LIN {X 0,Y 549.651,Z 687.436,A -85,B 0,C 180,E1 21205.612,E2 21205.612} C_VEL
LIN {X 0,Y 543.222,Z 825.686,A -85,B 0,C 180,E1 21203.522,E2 21203.522} C_VEL
LIN {X 0,Y 540.973,Z 851.994,A -85,B 0,C 180,E1 21203.026,E2 21203.026} C_VEL
LIN {X 0,Y 537.634,Z 879.368,A -85,B 0,C 180,E1 21202.319,E2 21202.319} C_VEL
LIN {X 0,Y 534.444,Z 901.056,A -85,B 0,C 180,E1 21201.617,E2 21201.617} C_VEL
LIN {X 0,Y 531.01,Z 921.384,A -85,B 0,C 180,E1 21200.832,E2 21200.832} C_VEL
LIN {X 0,Y 527.002,Z 942.572,A -85,B 0,C 180,E1 21199.871,E2 21199.871} C_VEL
LIN {X 0,Y 521.583,Z 968.283,A -85,B 0,C 180,E1 21198.494,E2 21198.494} C_VEL
LIN {X 0,Y 516.27,Z 990.784,A -85,B 0,C 180,E1 21197.06,E2 21197.06} C_VEL
LIN {X 0,Y 511.706,Z 1008.978,A -85,B 0,C 180,E1 21195.736,E2 21195.736} C_VEL
LIN {X 0,Y 507.179,Z 1026.1,A -85,B 0,C 180,E1 21194.336,E2 21194.336} C_VEL
LIN {X 0,Y 502.54,Z 1042.949,A -85,B 0,C 180,E1 21192.793,E2 21192.793} C_VEL
LIN {X 0,Y 497.445,Z 1060.954,A -85,B 0,C 180,E1 21190.939,E2 21190.939} C_VEL
LIN {X 0,Y 491.162,Z 1082.539,A -85,B 0,C 180,E1 21188.381,E2 21188.381} C_VEL
LIN {X 0,Y 486.635,Z 1097.975,A -85,B 0,C 180,E1 21186.28,E2 21186.28} C_VEL
LIN {X 0,Y 482.591,Z 1111.902,A -85,B 0,C 180,E1 21184.158,E2 21184.158} C_VEL
LIN {X 0,Y 479.016,Z 1124.472,A -85,B 0,C 180,E1 21182.017,E2 21182.017} C_VEL
LIN {X 0,Y 475.599,Z 1137.117,A -85,B 0,C 180,E1 21179.607,E2 21179.607} C_VEL
LIN {X 0,Y 472.036,Z 1151.255,A -85,B 0,C 180,E1 21176.547,E2 21176.547} C_VEL
LIN {X 0,Y 469.365,Z 1162.835,A -85,B 0,C 180,E1 21173.608,E2 21173.608} C_VEL
LIN {X 0,Y 467.505,Z 1172.064,A -85,B 0,C 180,E1 21170.926,E2 21170.926} C_VEL
LIN {X 0,Y 466.177,Z 1179.694,A -85,B 0,C 180,E1 21168.378,E2 21168.378} C_VEL
LIN {X 0,Y 465.207,Z 1186.55,A -85,B 0,C 180,E1 21165.712,E2 21165.712} C_VEL
LIN {X 0,Y 464.466,Z 1193.301,A -85,B 0,C 180,E1 21162.558,E2 21162.558} C_VEL
LIN {X 0,Y 464.091,Z 1198.542,A -85,B 0,C 180,E1 21159.299,E2 21159.299} C_VEL
LIN {X 0,Y 463.959,Z 1201.757,A -85,B 0,C 180,E1 21156.527,E2 21156.527} C_VEL
LIN {X 0,Y 463.915,Z 1203.743,A -85,B 0,C 180,E1 21153.955,E2 21153.955} C_VEL
LIN {X 0,Y 463.911,Z 1204.734,A -85,B 0,C 180,E1 21151.482,E2 21151.482} C_VEL
LIN {X 0,Y 463.908,Z 1204.825,A -85,B 0,C 180,E1 21149.012,E2 21149.012} C_VEL
LIN {X 0,Y 463.915,Z 1204.015,A -85,B 0,C 180,E1 21146.54,E2 21146.54} C_VEL
LIN {X 0,Y 463.947,Z 1202.181,A -85,B 0,C 180,E1 21143.938,E2 21143.938} C_VEL
LIN {X 0,Y 464.044,Z 1199.499,A -85,B 0,C 180,E1 21141.45,E2 21141.45} C_VEL
LIN {X 0,Y 464.248,Z 1195.868,A -85,B 0,C 180,E1 21138.949,E2 21138.949} C_VEL
LIN {X 0,Y 464.693,Z 1190.99,A -85,B 0,C 180,E1 21136.309,E2 21136.309} C_VEL
LIN {X 0,Y 465.387,Z 1185.014,A -85,B 0,C 180,E1 21133.653,E2 21133.653} C_VEL
LIN {X 0,Y 466.671,Z 1176.831,A -85,B 0,C 180,E1 21130.604,E2 21130.604} C_VEL
LIN {X 0,Y 468.694,Z 1166.058,A -85,B 0,C 180,E1 21127.287,E2 21127.287} C_VEL
LIN {X 0,Y 470.899,Z 1155.903,A -85,B 0,C 180,E1 21124.602,E2 21124.602} C_VEL
LIN {X 0,Y 473.407,Z 1145.514,A -85,B 0,C 180,E1 21122.176,E2 21122.176} C_VEL
LIN {X 0,Y 476.604,Z 1133.238,A -85,B 0,C 180,E1 21119.63,E2 21119.63} C_VEL
LIN {X 0,Y 481.3,Z 1116.533,A -85,B 0,C 180,E1 21116.598,E2 21116.598} C_VEL
LIN {X 0,Y 485.893,Z 1100.648,A -85,B 0,C 180,E1 21114.094,E2 21114.094} C_VEL
LIN {X 0,Y 490.368,Z 1085.693,A -85,B 0,C 180,E1 21111.992,E2 21111.992} C_VEL
LIN {X 0,Y 495.392,Z 1069.058,A -85,B 0,C 180,E1 21109.904,E2 21109.904} C_VEL
LIN {X 0,Y 501.937,Z 1047.349,A -85,B 0,C 180,E1 21107.524,E2 21107.524} C_VEL
LIN {X 0,Y 507.495,Z 1028.134,A -85,B 0,C 180,E1 21105.699,E2 21105.699} C_VEL
LIN {X 0,Y 512.508,Z 1010.266,A -85,B 0,C 180,E1 21104.196,E2 21104.196} C_VEL
LIN {X 0,Y 517.402,Z 991.974,A -85,B 0,C 180,E1 21102.831,E2 21102.831} C_VEL
LIN {X 0,Y 522.564,Z 971.525,A -85,B 0,C 180,E1 21101.489,E2 21101.489} C_VEL
LIN {X 0,Y 528.704,Z 945.004,A -85,B 0,C 180,E1 21100.012,E2 21100.012} C_VEL
LIN {X 0,Y 533.198,Z 923.023,A -85,B 0,C 180,E1 21098.988,E2 21098.988} C_VEL
LIN {X 0,Y 536.991,Z 902.347,A -85,B 0,C 180,E1 21098.171,E2 21098.171} C_VEL
LIN {X 0,Y 540.352,Z 881.367,A -85,B 0,C 180,E1 21097.475,E2 21097.475} C_VEL
LIN {X 0,Y 543.373,Z 859.139,A -85,B 0,C 180,E1 21096.872,E2 21096.872} C_VEL
LIN {X 0,Y 546.347,Z 831.001,A -85,B 0,C 180,E1 21096.29,E2 21096.29} C_VEL
LIN {X 0,Y 549.102,Z 782.806,A -85,B 0,C 180,E1 21095.529,E2 21095.529} C_VEL
LIN {X 0,Y 560.963,Z 560.073,A -85,B 0,C 180,E1 21092.109,E2 21092.109} C_VEL
LIN {X 0,Y 565.673,Z 475.855,A -85,B 0,C 180,E1 21090.8,E2 21090.8} C_VEL
LIN {X 0,Y 556.142,Z 460.846,A -85,B 0,C 180,E1 21088.483,E2 21088.483} C_VEL
LIN {X 0,Y 548.365,Z 449.512,A -85,B 0,C 180,E1 21086.389,E2 21086.389} C_VEL
LIN {X 0,Y 541.388,Z 439.723,A -85,B 0,C 180,E1 21084.293,E2 21084.293} C_VEL
LIN {X 0,Y 536.871,Z 433.476,A -85,B 0,C 180,E1 21082.792,E2 21082.792} C_VEL
LIN {X 0,Y 532.572,Z 428.076,A -85,B 0,C 180,E1 21081.245,E2 21081.245} C_VEL
LIN {X 0,Y 528.819,Z 423.299,A -85,B 0,C 180,E1 21079.754,E2 21079.754} C_VEL
LIN {X 0,Y 524.766,Z 418.77,A -85,B 0,C 180,E1 21077.979,E2 21077.979} C_VEL
LIN {X 0,Y 523.478,Z 416.816,A -85,B 0,C 180,E1 21077.336,E2 21077.336} C_VEL
LIN {X 0,Y 519.967,Z 413.289,A -85,B 0,C 180,E1 21075.503,E2 21075.503} C_VEL
LIN {X 0,Y 518.406,Z 410.788,A -85,B 0,C 180,E1 21074.521,E2 21074.521} C_VEL
LIN {X 0,Y 515.036,Z 407.8,A -85,B 0,C 180,E1 21072.217,E2 21072.217} C_VEL
LIN {X 0,Y 513.302,Z 404.463,A -85,B 0,C 180,E1 21070.551,E2 21070.551} C_VEL
LIN {X 0,Y 509.592,Z 401.905,A -85,B 0,C 180,E1 21064.276,E2 21064.276} C_VEL
LIN {X 0,Y 509.876,Z 402.177,A -85,B 0,C 180,E1 21061.236,E2 21061.236} C_VEL
LIN {X 0,Y 513.509,Z 404.739,A -85,B 0,C 180,E1 21056.036,E2 21056.036} C_VEL
LIN {X 0,Y 515.352,Z 408.233,A -85,B 0,C 180,E1 21054.321,E2 21054.321} C_VEL
LIN {X 0,Y 518.812,Z 411.217,A -85,B 0,C 180,E1 21052.024,E2 21052.024} C_VEL
LIN {X 0,Y 521.465,Z 415.141,A -85,B 0,C 180,E1 21050.453,E2 21050.453} C_VEL
LIN {X 0,Y 524.069,Z 417.551,A -85,B 0,C 180,E1 21049.168,E2 21049.168} C_VEL
LIN {X 0,Y 527.266,Z 421.812,A -85,B 0,C 180,E1 21047.682,E2 21047.682} C_VEL
LIN {X 0,Y 529.035,Z 423.657,A -85,B 0,C 180,E1 21046.947,E2 21046.947} C_VEL
LIN {X 0,Y 532.738,Z 428.24,A -85,B 0,C 180,E1 21045.489,E2 21045.489} C_VEL
LIN {X 0,Y 538.696,Z 435.728,A -85,B 0,C 180,E1 21043.391,E2 21043.391} C_VEL
LIN {X 0,Y 543.283,Z 441.609,A -85,B 0,C 180,E1 21041.934,E2 21041.934} C_VEL
LIN {X 0,Y 549.857,Z 450.066,A -85,B 0,C 180,E1 21040.037,E2 21040.037} C_VEL
LIN {X 0,Y 559.197,Z 463.027,A -85,B 0,C 180,E1 21037.613,E2 21037.613} C_VEL
LIN {X 0,Y 565.694,Z 473.379,A -85,B 0,C 180,E1 21036.056,E2 21036.056} C_VEL
LIN {X 0,Y 553.81,Z 688.927,A -85,B 0,C 180,E1 21032.734,E2 21032.734} C_VEL
LIN {X 0,Y 546.853,Z 819.072,A -85,B 0,C 180,E1 21030.725,E2 21030.725} C_VEL
LIN {X 0,Y 544.343,Z 846.185,A -85,B 0,C 180,E1 21030.201,E2 21030.201} C_VEL
LIN {X 0,Y 540.821,Z 872.767,A -85,B 0,C 180,E1 21029.495,E2 21029.495} C_VEL
LIN {X 0,Y 537.599,Z 893.258,A -85,B 0,C 180,E1 21028.819,E2 21028.819} C_VEL
LIN {X 0,Y 533.943,Z 913.499,A -85,B 0,C 180,E1 21028.025,E2 21028.025} C_VEL
LIN {X 0,Y 529.736,Z 934.282,A -85,B 0,C 180,E1 21027.07,E2 21027.07} C_VEL
LIN {X 0,Y 524.349,Z 958.432,A -85,B 0,C 180,E1 21025.768,E2 21025.768} C_VEL
LIN {X 0,Y 518.322,Z 982.281,A -85,B 0,C 180,E1 21024.231,E2 21024.231} C_VEL
LIN {X 0,Y 513.236,Z 1001.222,A -85,B 0,C 180,E1 21022.824,E2 21022.824} C_VEL
LIN {X 0,Y 508.27,Z 1018.81,A -85,B 0,C 180,E1 21021.349,E2 21021.349} C_VEL
LIN {X 0,Y 503.044,Z 1036.665,A -85,B 0,C 180,E1 21019.663,E2 21019.663} C_VEL
LIN {X 0,Y 496.66,Z 1057.893,A -85,B 0,C 180,E1 21017.376,E2 21017.376} C_VEL
LIN {X 0,Y 491.067,Z 1075.973,A -85,B 0,C 180,E1 21015.118,E2 21015.118} C_VEL
LIN {X 0,Y 486.515,Z 1090.867,A -85,B 0,C 180,E1 21013.024,E2 21013.024} C_VEL
LIN {X 0,Y 482.248,Z 1105.162,A -85,B 0,C 180,E1 21010.775,E2 21010.775} C_VEL
LIN {X 0,Y 477.553,Z 1121.65,A -85,B 0,C 180,E1 21007.84,E2 21007.84} C_VEL
LIN {X 0,Y 475.09,Z 1130.636,A -85,B 0,C 180,E1 21006.035,E2 21006.035} C_VEL
LIN {X 0,Y 473.128,Z 1134.565,A -85,B 0,C 180,E1 21005.261,E2 21005.261} C_VEL
LIN {X 0,Y 464.651,Z 1144.816,A -85,B 0,C 180,E1 21003.232,E2 21003.232} C_VEL
LIN {X 0,Y 463.204,Z 1147.79,A -85,B 0,C 180,E1 21002.52,E2 21002.52} C_VEL
LIN {X 0,Y 460.393,Z 1159.963,A -85,B 0,C 180,E1 20999.109,E2 20999.109} C_VEL
LIN {X 0,Y 458.412,Z 1169.958,A -85,B 0,C 180,E1 20995.725,E2 20995.725} C_VEL
LIN {X 0,Y 457.267,Z 1177.255,A -85,B 0,C 180,E1 20992.77,E2 20992.77} C_VEL
LIN {X 0,Y 456.495,Z 1183.735,A -85,B 0,C 180,E1 20989.579,E2 20989.579} C_VEL
LIN {X 0,Y 456.092,Z 1188.961,A -85,B 0,C 180,E1 20986.165,E2 20986.165} C_VEL
LIN {X 0,Y 455.953,Z 1192.065,A -85,B 0,C 180,E1 20983.312,E2 20983.312} C_VEL
LIN {X 0,Y 455.916,Z 1193.909,A -85,B 0,C 180,E1 20980.724,E2 20980.724} C_VEL
LIN {X 0,Y 455.908,Z 1194.803,A -85,B 0,C 180,E1 20978.196,E2 20978.196} C_VEL
LIN {X 0,Y 455.911,Z 1194.794,A -85,B 0,C 180,E1 20975.664,E2 20975.664} C_VEL
LIN {X 0,Y 455.916,Z 1193.822,A -85,B 0,C 180,E1 20973.017,E2 20973.017} C_VEL
LIN {X 0,Y 455.974,Z 1191.657,A -85,B 0,C 180,E1 20970.126,E2 20970.126} C_VEL
LIN {X 0,Y 456.177,Z 1187.597,A -85,B 0,C 180,E1 20966.733,E2 20966.733} C_VEL
LIN {X 0,Y 456.608,Z 1182.552,A -85,B 0,C 180,E1 20963.714,E2 20963.714} C_VEL
LIN {X 0,Y 457.356,Z 1176.516,A -85,B 0,C 180,E1 20960.817,E2 20960.817} C_VEL
LIN {X 0,Y 458.685,Z 1168.537,A -85,B 0,C 180,E1 20957.665,E2 20957.665} C_VEL
LIN {X 0,Y 460.867,Z 1157.701,A -85,B 0,C 180,E1 20954.136,E2 20954.136} C_VEL
LIN {X 0,Y 463.467,Z 1146.69,A -85,B 0,C 180,E1 20951.119,E2 20951.119} C_VEL
LIN {X 0,Y 466.481,Z 1135.156,A -85,B 0,C 180,E1 20948.367,E2 20948.367} C_VEL
LIN {X 0,Y 470.784,Z 1120.249,A -85,B 0,C 180,E1 20945.267,E2 20945.267} C_VEL
LIN {X 0,Y 475.265,Z 1105.063,A -85,B 0,C 180,E1 20942.566,E2 20942.566} C_VEL
LIN {X 0,Y 479.518,Z 1091.202,A -85,B 0,C 180,E1 20940.385,E2 20940.385} C_VEL
LIN {X 0,Y 484.266,Z 1075.83,A -85,B 0,C 180,E1 20938.231,E2 20938.231} C_VEL
LIN {X 0,Y 490.176,Z 1056.8,A -85,B 0,C 180,E1 20935.879,E2 20935.879} C_VEL
LIN {X 0,Y 496.306,Z 1036.036,A -85,B 0,C 180,E1 20933.68,E2 20933.68} C_VEL
LIN {X 0,Y 501.213,Z 1018.99,A -85,B 0,C 180,E1 20932.09,E2 20932.09} C_VEL
LIN {X 0,Y 506.037,Z 1001.468,A -85,B 0,C 180,E1 20930.636,E2 20930.636} C_VEL
LIN {X 0,Y 510.938,Z 982.649,A -85,B 0,C 180,E1 20929.253,E2 20929.253} C_VEL
LIN {X 0,Y 516.7,Z 959.081,A -85,B 0,C 180,E1 20927.744,E2 20927.744} C_VEL
LIN {X 0,Y 521.835,Z 935.199,A -85,B 0,C 180,E1 20926.464,E2 20926.464} C_VEL
LIN {X 0,Y 525.854,Z 914.588,A -85,B 0,C 180,E1 20925.52,E2 20925.52} C_VEL
LIN {X 0,Y 529.423,Z 894.057,A -85,B 0,C 180,E1 20924.718,E2 20924.718} C_VEL
LIN {X 0,Y 532.612,Z 872.81,A -85,B 0,C 180,E1 20924.019,E2 20924.019} C_VEL
LIN {X 0,Y 535.973,Z 846.163,A -85,B 0,C 180,E1 20923.314,E2 20923.314} C_VEL
LIN {X 0,Y 538.366,Z 818.867,A -85,B 0,C 180,E1 20922.792,E2 20922.792} C_VEL
LIN {X 0,Y 544.33,Z 695.866,A -85,B 0,C 180,E1 20920.922,E2 20920.922} C_VEL
LIN {X 0,Y 555.064,Z 476.693,A -85,B 0,C 180,E1 20917.593,E2 20917.593} C_VEL
LIN {X 0,Y 554.881,Z 475.782,A -85,B 0,C 180,E1 20917.543,E2 20917.543} C_VEL
LIN {X 0,Y 544.972,Z 460.83,A -85,B 0,C 180,E1 20915.532,E2 20915.532} C_VEL
LIN {X 0,Y 533.991,Z 445.737,A -85,B 0,C 180,E1 20913.114,E2 20913.114} C_VEL
LIN {X 0,Y 525.45,Z 434.579,A -85,B 0,C 180,E1 20911.044,E2 20911.044} C_VEL
LIN {X 0,Y 518.137,Z 425.158,A -85,B 0,C 180,E1 20909.098,E2 20909.098} C_VEL
LIN {X 0,Y 513.762,Z 419.766,A -85,B 0,C 180,E1 20907.846,E2 20907.846} C_VEL
LIN {X 0,Y 509.435,Z 414.406,A -85,B 0,C 180,E1 20906.521,E2 20906.521} C_VEL
LIN {X 0,Y 504.85,Z 408.87,A -85,B 0,C 180,E1 20905.015,E2 20905.015} C_VEL
LIN {X 0,Y 501.142,Z 404.499,A -85,B 0,C 180,E1 20903.7,E2 20903.7} C_VEL
LIN {X 0,Y 499.827,Z 402.982,A -85,B 0,C 180,E1 20903.21,E2 20903.21} C_VEL
LIN {X 0,Y 496.356,Z 399.083,A -85,B 0,C 180,E1 20901.85,E2 20901.85} C_VEL
LIN {X 0,Y 495.128,Z 397.19,A -85,B 0,C 180,E1 20901.316,E2 20901.316} C_VEL
LIN {X 0,Y 491.632,Z 393.913,A -85,B 0,C 180,E1 20899.794,E2 20899.794} C_VEL
LIN {X 0,Y 489.71,Z 390.934,A -85,B 0,C 180,E1 20898.821,E2 20898.821} C_VEL
LIN {X 0,Y 486.447,Z 388.452,A -85,B 0,C 180,E1 20897.155,E2 20897.155} C_VEL
LIN {X 0,Y 484.363,Z 384.721,A -85,B 0,C 180,E1 20895.813,E2 20895.813} C_VEL
LIN {X 0,Y 480.409,Z 381.967,A -85,B 0,C 180,E1 20893.113,E2 20893.113} C_VEL
LIN {X 0,Y 478.502,Z 378.278,A -85,B 0,C 180,E1 20891.206,E2 20891.206} C_VEL
LIN {X 0,Y 478.048,Z 377.801,A -85,B 0,C 180,E1 20890.728,E2 20890.728} C_VEL
LIN {X 0,Y 474.633,Z 375.968,A -85,B 0,C 180,E1 20884.228,E2 20884.228} C_VEL
LIN {X 0,Y 475.297,Z 376.512,A -85,B 0,C 180,E1 20880.241,E2 20880.241} C_VEL
LIN {X 0,Y 478.483,Z 378.16,A -85,B 0,C 180,E1 20875.926,E2 20875.926} C_VEL
LIN {X 0,Y 480.364,Z 381.936,A -85,B 0,C 180,E1 20874.026,E2 20874.026} C_VEL
LIN {X 0,Y 484.421,Z 384.931,A -85,B 0,C 180,E1 20871.244,E2 20871.244} C_VEL
LIN {X 0,Y 486.469,Z 388.438,A -85,B 0,C 180,E1 20869.938,E2 20869.938} C_VEL
LIN {X 0,Y 490.121,Z 391.389,A -85,B 0,C 180,E1 20868.079,E2 20868.079} C_VEL
LIN {X 0,Y 492.974,Z 395.508,A -85,B 0,C 180,E1 20866.69,E2 20866.69} C_VEL
LIN {X 0,Y 495.56,Z 397.796,A -85,B 0,C 180,E1 20865.6,E2 20865.6} C_VEL
LIN {X 0,Y 498.739,Z 402.022,A -85,B 0,C 180,E1 20864.297,E2 20864.297} C_VEL
LIN {X 0,Y 500.891,Z 404.06,A -85,B 0,C 180,E1 20863.503,E2 20863.503} C_VEL
LIN {X 0,Y 504.6,Z 408.613,A -85,B 0,C 180,E1 20862.173,E2 20862.173} C_VEL
LIN {X 0,Y 506.266,Z 410.618,A -85,B 0,C 180,E1 20861.608,E2 20861.608} C_VEL
LIN {X 0,Y 511.081,Z 416.441,A -85,B 0,C 180,E1 20860.068,E2 20860.068} C_VEL
LIN {X 0,Y 516.19,Z 422.736,A -85,B 0,C 180,E1 20858.554,E2 20858.554} C_VEL
LIN {X 0,Y 521.204,Z 429.022,A -85,B 0,C 180,E1 20857.17,E2 20857.17} C_VEL
LIN {X 0,Y 528.614,Z 439.045,A -85,B 0,C 180,E1 20855.26,E2 20855.26} C_VEL
LIN {X 0,Y 539.958,Z 455.564,A -85,B 0,C 180,E1 20852.602,E2 20852.602} C_VEL
LIN {X 0,Y 552.93,Z 475.552,A -85,B 0,C 180,E1 20849.88,E2 20849.88} C_VEL
LIN {X 0,Y 555.066,Z 479.191,A -85,B 0,C 180,E1 20849.453,E2 20849.453} C_VEL
LIN {X 0,Y 544.676,Z 691.913,A -85,B 0,C 180,E1 20846.221,E2 20846.221} C_VEL
LIN {X 0,Y 538.232,Z 825.714,A -85,B 0,C 180,E1 20844.188,E2 20844.188} C_VEL
LIN {X 0,Y 535.869,Z 852.634,A -85,B 0,C 180,E1 20843.678,E2 20843.678} C_VEL
LIN {X 0,Y 532.469,Z 879.552,A -85,B 0,C 180,E1 20842.978,E2 20842.978} C_VEL
LIN {X 0,Y 529.193,Z 901.157,A -85,B 0,C 180,E1 20842.276,E2 20842.276} C_VEL
LIN {X 0,Y 525.597,Z 921.833,A -85,B 0,C 180,E1 20841.474,E2 20841.474} C_VEL
LIN {X 0,Y 521.474,Z 942.982,A -85,B 0,C 180,E1 20840.51,E2 20840.51} C_VEL
LIN {X 0,Y 515.816,Z 968.907,A -85,B 0,C 180,E1 20839.11,E2 20839.11} C_VEL
LIN {X 0,Y 510.472,Z 990.866,A -85,B 0,C 180,E1 20837.702,E2 20837.702} C_VEL
LIN {X 0,Y 505.707,Z 1009.256,A -85,B 0,C 180,E1 20836.355,E2 20836.355} C_VEL
LIN {X 0,Y 501.026,Z 1026.358,A -85,B 0,C 180,E1 20834.947,E2 20834.947} C_VEL
LIN {X 0,Y 495.943,Z 1044.189,A -85,B 0,C 180,E1 20833.295,E2 20833.295} C_VEL
LIN {X 0,Y 489.829,Z 1065.1,A -85,B 0,C 180,E1 20831.092,E2 20831.092} C_VEL
LIN {X 0,Y 483.991,Z 1084.163,A -85,B 0,C 180,E1 20828.752,E2 20828.752} C_VEL
LIN {X 0,Y 479.602,Z 1098.623,A -85,B 0,C 180,E1 20826.75,E2 20826.75} C_VEL
LIN {X 0,Y 475.404,Z 1112.517,A -85,B 0,C 180,E1 20824.601,E2 20824.601} C_VEL
LIN {X 0,Y 471.263,Z 1126.56,A -85,B 0,C 180,E1 20822.159,E2 20822.159} C_VEL
LIN {X 0,Y 466.786,Z 1142.559,A -85,B 0,C 180,E1 20818.953,E2 20818.953} C_VEL
LIN {X 0,Y 463.732,Z 1154.271,A -85,B 0,C 180,E1 20816.232,E2 20816.232} C_VEL
LIN {X 0,Y 461.405,Z 1164.129,A -85,B 0,C 180,E1 20813.634,E2 20813.634} C_VEL
LIN {X 0,Y 459.589,Z 1172.789,A -85,B 0,C 180,E1 20811.037,E2 20811.037} C_VEL
LIN {X 0,Y 458.102,Z 1181.027,A -85,B 0,C 180,E1 20808.187,E2 20808.187} C_VEL
LIN {X 0,Y 456.901,Z 1189.62,A -85,B 0,C 180,E1 20804.576,E2 20804.576} C_VEL
LIN {X 0,Y 456.323,Z 1195.154,A -85,B 0,C 180,E1 20801.629,E2 20801.629} C_VEL
LIN {X 0,Y 456.077,Z 1198.95,A -85,B 0,C 180,E1 20799.082,E2 20799.082} C_VEL
LIN {X 0,Y 455.96,Z 1201.798,A -85,B 0,C 180,E1 20796.548,E2 20796.548} C_VEL
LIN {X 0,Y 455.915,Z 1203.718,A -85,B 0,C 180,E1 20794.024,E2 20794.024} C_VEL
LIN {X 0,Y 455.91,Z 1204.722,A -85,B 0,C 180,E1 20791.508,E2 20791.508} C_VEL
LIN {X 0,Y 455.908,Z 1204.814,A -85,B 0,C 180,E1 20788.995,E2 20788.995} C_VEL
LIN {X 0,Y 455.915,Z 1203.992,A -85,B 0,C 180,E1 20786.479,E2 20786.479} C_VEL
LIN {X 0,Y 455.946,Z 1202.255,A -85,B 0,C 180,E1 20783.958,E2 20783.958} C_VEL
LIN {X 0,Y 456.046,Z 1199.592,A -85,B 0,C 180,E1 20781.426,E2 20781.426} C_VEL
LIN {X 0,Y 456.257,Z 1195.985,A -85,B 0,C 180,E1 20778.881,E2 20778.881} C_VEL
LIN {X 0,Y 456.723,Z 1191.154,A -85,B 0,C 180,E1 20776.195,E2 20776.195} C_VEL
LIN {X 0,Y 457.405,Z 1185.531,A -85,B 0,C 180,E1 20773.621,E2 20773.621} C_VEL
LIN {X 0,Y 458.53,Z 1178.517,A -85,B 0,C 180,E1 20770.908,E2 20770.908} C_VEL
LIN {X 0,Y 460.416,Z 1168.767,A -85,B 0,C 180,E1 20767.692,E2 20767.692} C_VEL
LIN {X 0,Y 463.097,Z 1156.839,A -85,B 0,C 180,E1 20764.417,E2 20764.417} C_VEL
LIN {X 0,Y 465.832,Z 1145.987,A -85,B 0,C 180,E1 20761.822,E2 20761.822} C_VEL
LIN {X 0,Y 469.183,Z 1133.788,A -85,B 0,C 180,E1 20759.239,E2 20759.239} C_VEL
LIN {X 0,Y 473.992,Z 1117.592,A -85,B 0,C 180,E1 20756.217,E2 20756.217} C_VEL
LIN {X 0,Y 479.126,Z 1100.682,A -85,B 0,C 180,E1 20753.505,E2 20753.505} C_VEL
LIN {X 0,Y 483.84,Z 1085.664,A -85,B 0,C 180,E1 20751.368,E2 20751.368} C_VEL
LIN {X 0,Y 489.017,Z 1069.294,A -85,B 0,C 180,E1 20749.29,E2 20749.29} C_VEL
LIN {X 0,Y 495.701,Z 1048.091,A -85,B 0,C 180,E1 20746.931,E2 20746.931} C_VEL
LIN {X 0,Y 501.825,Z 1027.732,A -85,B 0,C 180,E1 20744.983,E2 20744.983} C_VEL
LIN {X 0,Y 506.942,Z 1010.177,A -85,B 0,C 180,E1 20743.501,E2 20743.501} C_VEL
LIN {X 0,Y 511.9,Z 992.339,A -85,B 0,C 180,E1 20742.162,E2 20742.162} C_VEL
LIN {X 0,Y 516.998,Z 972.844,A -85,B 0,C 180,E1 20740.872,E2 20740.872} C_VEL
LIN {X 0,Y 523.101,Z 947.813,A -85,B 0,C 180,E1 20739.448,E2 20739.448} C_VEL
LIN {X 0,Y 528.2,Z 923.725,A -85,B 0,C 180,E1 20738.314,E2 20738.314} C_VEL
LIN {X 0,Y 532.216,Z 902.511,A -85,B 0,C 180,E1 20737.473,E2 20737.473} C_VEL
LIN {X 0,Y 535.73,Z 881.253,A -85,B 0,C 180,E1 20736.768,E2 20736.768} C_VEL
LIN {X 0,Y 538.824,Z 859.122,A -85,B 0,C 180,E1 20736.168,E2 20736.168} C_VEL
LIN {X 0,Y 541.895,Z 830.906,A -85,B 0,C 180,E1 20735.584,E2 20735.584} C_VEL
LIN {X 0,Y 544.71,Z 783.337,A -85,B 0,C 180,E1 20734.83,E2 20734.83} C_VEL
LIN {X 0,Y 556.987,Z 560.731,A -85,B 0,C 180,E1 20731.4,E2 20731.4} C_VEL
LIN {X 0,Y 561.59,Z 480.363,A -85,B 0,C 180,E1 20730.139,E2 20730.139} C_VEL
LIN {X 0,Y 552.729,Z 466.423,A -85,B 0,C 180,E1 20727.91,E2 20727.91} C_VEL
LIN {X 0,Y 545.838,Z 456.154,A -85,B 0,C 180,E1 20725.994,E2 20725.994} C_VEL
LIN {X 0,Y 537.556,Z 444.253,A -85,B 0,C 180,E1 20723.399,E2 20723.399} C_VEL
LIN {X 0,Y 530.921,Z 435.642,A -85,B 0,C 180,E1 20721.025,E2 20721.025} C_VEL
LIN {X 0,Y 526.526,Z 430.185,A -85,B 0,C 180,E1 20719.237,E2 20719.237} C_VEL
LIN {X 0,Y 523.025,Z 425.982,A -85,B 0,C 180,E1 20717.639,E2 20717.639} C_VEL
LIN {X 0,Y 522.076,Z 424.547,A -85,B 0,C 180,E1 20717.154,E2 20717.154} C_VEL
LIN {X 0,Y 518.536,Z 420.853,A -85,B 0,C 180,E1 20715.261,E2 20715.261} C_VEL
LIN {X 0,Y 517.268,Z 418.675,A -85,B 0,C 180,E1 20714.44,E2 20714.44} C_VEL
LIN {X 0,Y 513.928,Z 415.7,A -85,B 0,C 180,E1 20712.13,E2 20712.13} C_VEL
LIN {X 0,Y 512.217,Z 412.375,A -85,B 0,C 180,E1 20710.46,E2 20710.46} C_VEL
LIN {X 0,Y 508.616,Z 409.847,A -85,B 0,C 180,E1 20704.284,E2 20704.284} C_VEL
LIN {X 0,Y 508.896,Z 410.125,A -85,B 0,C 180,E1 20701.238,E2 20701.238} C_VEL
LIN {X 0,Y 512.353,Z 412.559,A -85,B 0,C 180,E1 20696.195,E2 20696.195} C_VEL
LIN {X 0,Y 514.226,Z 416.108,A -85,B 0,C 180,E1 20694.421,E2 20694.421} C_VEL
LIN {X 0,Y 517.551,Z 419.077,A -85,B 0,C 180,E1 20692.172,E2 20692.172} C_VEL
LIN {X 0,Y 520.379,Z 423.132,A -85,B 0,C 180,E1 20690.488,E2 20690.488} C_VEL
LIN {X 0,Y 522.633,Z 425.262,A -85,B 0,C 180,E1 20689.361,E2 20689.361} C_VEL
LIN {X 0,Y 526.036,Z 429.72,A -85,B 0,C 180,E1 20687.764,E2 20687.764} C_VEL
LIN {X 0,Y 527.528,Z 431.384,A -85,B 0,C 180,E1 20687.132,E2 20687.132} C_VEL
LIN {X 0,Y 531.476,Z 436.166,A -85,B 0,C 180,E1 20685.565,E2 20685.565} C_VEL
LIN {X 0,Y 537.077,Z 443.488,A -85,B 0,C 180,E1 20683.562,E2 20683.562} C_VEL
LIN {X 0,Y 541.381,Z 449.056,A -85,B 0,C 180,E1 20682.174,E2 20682.174} C_VEL
LIN {X 0,Y 547.782,Z 457.44,A -85,B 0,C 180,E1 20680.292,E2 20680.292} C_VEL
LIN {X 0,Y 556.727,Z 470.011,A -85,B 0,C 180,E1 20677.925,E2 20677.925} C_VEL
LIN {X 0,Y 561.662,Z 477.995,A -85,B 0,C 180,E1 20676.707,E2 20676.707} C_VEL
LIN {X 0,Y 549.263,Z 695.541,A -85,B 0,C 180,E1 20673.345,E2 20673.345} C_VEL
LIN {X 0,Y 542.419,Z 819.153,A -85,B 0,C 180,E1 20671.429,E2 20671.429} C_VEL
LIN {X 0,Y 539.835,Z 846.294,A -85,B 0,C 180,E1 20670.904,E2 20670.904} C_VEL
LIN {X 0,Y 536.215,Z 872.836,A -85,B 0,C 180,E1 20670.2,E2 20670.2} C_VEL
LIN {X 0,Y 532.859,Z 893.525,A -85,B 0,C 180,E1 20669.517,E2 20669.517} C_VEL
LIN {X 0,Y 529.085,Z 913.805,A -85,B 0,C 180,E1 20668.721,E2 20668.721} C_VEL
LIN {X 0,Y 524.679,Z 934.861,A -85,B 0,C 180,E1 20667.751,E2 20667.751} C_VEL
LIN {X 0,Y 519.092,Z 959.063,A -85,B 0,C 180,E1 20666.439,E2 20666.439} C_VEL
LIN {X 0,Y 512.823,Z 982.961,A -85,B 0,C 180,E1 20664.887,E2 20664.887} C_VEL
LIN {X 0,Y 507.59,Z 1001.729,A -85,B 0,C 180,E1 20663.483,E2 20663.483} C_VEL
LIN {X 0,Y 502.446,Z 1019.268,A -85,B 0,C 180,E1 20662.002,E2 20662.002} C_VEL
LIN {X 0,Y 497.02,Z 1037.059,A -85,B 0,C 180,E1 20660.307,E2 20660.307} C_VEL
LIN {X 0,Y 490.209,Z 1058.738,A -85,B 0,C 180,E1 20657.939,E2 20657.939} C_VEL
LIN {X 0,Y 484.555,Z 1076.236,A -85,B 0,C 180,E1 20655.727,E2 20655.727} C_VEL
LIN {X 0,Y 479.71,Z 1091.374,A -85,B 0,C 180,E1 20653.569,E2 20653.569} C_VEL
LIN {X 0,Y 475.078,Z 1106.137,A -85,B 0,C 180,E1 20651.204,E2 20651.204} C_VEL
LIN {X 0,Y 469.765,Z 1123.746,A -85,B 0,C 180,E1 20647.96,E2 20647.96} C_VEL
LIN {X 0,Y 466.294,Z 1135.921,A -85,B 0,C 180,E1 20645.377,E2 20645.377} C_VEL
LIN {X 0,Y 463.372,Z 1147.104,A -85,B 0,C 180,E1 20642.694,E2 20642.694} C_VEL
LIN {X 0,Y 463.204,Z 1147.79,A -85,B 0,C 180,E1 20642.52,E2 20642.52} C_VEL
LIN {X 0,Y 461.445,Z 1151.24,A -85,B 0,C 180,E1 20641.683,E2 20641.683} C_VEL
LIN {X 0,Y 453.433,Z 1160.012,A -85,B 0,C 180,E1 20639.473,E2 20639.473} C_VEL
LIN {X 0,Y 452.142,Z 1162.468,A -85,B 0,C 180,E1 20638.708,E2 20638.708} C_VEL
LIN {X 0,Y 450.464,Z 1170.765,A -85,B 0,C 180,E1 20635.788,E2 20635.788} C_VEL
LIN {X 0,Y 449.249,Z 1178.263,A -85,B 0,C 180,E1 20632.646,E2 20632.646} C_VEL
LIN {X 0,Y 448.438,Z 1184.962,A -85,B 0,C 180,E1 20629.133,E2 20629.133} C_VEL
LIN {X 0,Y 448.09,Z 1189.374,A -85,B 0,C 180,E1 20626.063,E2 20626.063} C_VEL
LIN {X 0,Y 447.954,Z 1192.271,A -85,B 0,C 180,E1 20623.291,E2 20623.291} C_VEL
LIN {X 0,Y 447.917,Z 1194.057,A -85,B 0,C 180,E1 20620.677,E2 20620.677} C_VEL
LIN {X 0,Y 447.905,Z 1194.913,A -85,B 0,C 180,E1 20618.085,E2 20618.085} C_VEL
LIN {X 0,Y 447.913,Z 1194.859,A -85,B 0,C 180,E1 20615.508,E2 20615.508} C_VEL
LIN {X 0,Y 447.919,Z 1193.779,A -85,B 0,C 180,E1 20612.687,E2 20612.687} C_VEL
LIN {X 0,Y 448.001,Z 1191.172,A -85,B 0,C 180,E1 20609.361,E2 20609.361} C_VEL
LIN {X 0,Y 448.246,Z 1186.903,A -85,B 0,C 180,E1 20606.035,E2 20606.035} C_VEL
LIN {X 0,Y 448.762,Z 1181.923,A -85,B 0,C 180,E1 20603.09,E2 20603.09} C_VEL
LIN {X 0,Y 449.667,Z 1175.429,A -85,B 0,C 180,E1 20600.012,E2 20600.012} C_VEL
LIN {X 0,Y 451.375,Z 1166.122,A -85,B 0,C 180,E1 20596.42,E2 20596.42} C_VEL
LIN {X 0,Y 453.604,Z 1156.034,A -85,B 0,C 180,E1 20593.217,E2 20593.217} C_VEL
LIN {X 0,Y 456.198,Z 1145.773,A -85,B 0,C 180,E1 20590.407,E2 20590.407} C_VEL
LIN {X 0,Y 459.315,Z 1134.677,A -85,B 0,C 180,E1 20587.743,E2 20587.743} C_VEL
LIN {X 0,Y 463.856,Z 1119.53,A -85,B 0,C 180,E1 20584.583,E2 20584.583} C_VEL
LIN {X 0,Y 468.353,Z 1105.051,A -85,B 0,C 180,E1 20581.988,E2 20581.988} C_VEL
LIN {X 0,Y 472.795,Z 1091.152,A -85,B 0,C 180,E1 20579.78,E2 20579.78} C_VEL
LIN {X 0,Y 477.449,Z 1076.635,A -85,B 0,C 180,E1 20577.723,E2 20577.723} C_VEL
LIN {X 0,Y 483.061,Z 1059.113,A -85,B 0,C 180,E1 20575.521,E2 20575.521} C_VEL
LIN {X 0,Y 489.82,Z 1037.241,A -85,B 0,C 180,E1 20573.15,E2 20573.15} C_VEL
LIN {X 0,Y 495.136,Z 1019.376,A -85,B 0,C 180,E1 20571.467,E2 20571.467} C_VEL
LIN {X 0,Y 500.121,Z 1001.86,A -85,B 0,C 180,E1 20570.003,E2 20570.003} C_VEL
LIN {X 0,Y 505.156,Z 983.144,A -85,B 0,C 180,E1 20568.617,E2 20568.617} C_VEL
LIN {X 0,Y 511.112,Z 959.512,A -85,B 0,C 180,E1 20567.096,E2 20567.096} C_VEL
LIN {X 0,Y 516.621,Z 934.591,A -85,B 0,C 180,E1 20565.757,E2 20565.757} C_VEL
LIN {X 0,Y 520.689,Z 914.279,A -85,B 0,C 180,E1 20564.828,E2 20564.828} C_VEL
LIN {X 0,Y 524.316,Z 893.92,A -85,B 0,C 180,E1 20564.034,E2 20564.034} C_VEL
LIN {X 0,Y 527.658,Z 872.184,A -85,B 0,C 180,E1 20563.321,E2 20563.321} C_VEL
LIN {X 0,Y 531.131,Z 844.871,A -85,B 0,C 180,E1 20562.608,E2 20562.608} C_VEL
LIN {X 0,Y 533.475,Z 818.636,A -85,B 0,C 180,E1 20562.109,E2 20562.109} C_VEL
LIN {X 0,Y 540.6,Z 675.831,A -85,B 0,C 180,E1 20559.929,E2 20559.929} C_VEL
LIN {X 0,Y 550.494,Z 480.4,A -85,B 0,C 180,E1 20556.944,E2 20556.944} C_VEL
LIN {X 0,Y 541.874,Z 467.292,A -85,B 0,C 180,E1 20555.15,E2 20555.15} C_VEL
LIN {X 0,Y 531.249,Z 452.512,A -85,B 0,C 180,E1 20552.76,E2 20552.76} C_VEL
LIN {X 0,Y 522.721,Z 441.238,A -85,B 0,C 180,E1 20550.649,E2 20550.649} C_VEL
LIN {X 0,Y 515.52,Z 431.904,A -85,B 0,C 180,E1 20548.689,E2 20548.689} C_VEL
LIN {X 0,Y 511.572,Z 426.958,A -85,B 0,C 180,E1 20547.533,E2 20547.533} C_VEL
LIN {X 0,Y 507.304,Z 421.627,A -85,B 0,C 180,E1 20546.2,E2 20546.2} C_VEL
LIN {X 0,Y 502.949,Z 416.292,A -85,B 0,C 180,E1 20544.739,E2 20544.739} C_VEL
LIN {X 0,Y 499.102,Z 411.575,A -85,B 0,C 180,E1 20543.339,E2 20543.339} C_VEL
LIN {X 0,Y 494.656,Z 406.568,A -85,B 0,C 180,E1 20541.586,E2 20541.586} C_VEL
LIN {X 0,Y 493.37,Z 404.732,A -85,B 0,C 180,E1 20541.022,E2 20541.022} C_VEL
LIN {X 0,Y 489.838,Z 401.149,A -85,B 0,C 180,E1 20539.433,E2 20539.433} C_VEL
LIN {X 0,Y 488.288,Z 398.703,A -85,B 0,C 180,E1 20538.63,E2 20538.63} C_VEL
LIN {X 0,Y 484.982,Z 396.033,A -85,B 0,C 180,E1 20536.9,E2 20536.9} C_VEL
LIN {X 0,Y 482.837,Z 392.367,A -85,B 0,C 180,E1 20535.494,E2 20535.494} C_VEL
LIN {X 0,Y 479.298,Z 389.864,A -85,B 0,C 180,E1 20533.021,E2 20533.021} C_VEL
LIN {X 0,Y 477.354,Z 386.151,A -85,B 0,C 180,E1 20531.05,E2 20531.05} C_VEL
LIN {X 0,Y 476.849,Z 385.685,A -85,B 0,C 180,E1 20530.511,E2 20530.511} C_VEL
LIN {X 0,Y 473.657,Z 383.909,A -85,B 0,C 180,E1 20524.237,E2 20524.237} C_VEL
LIN {X 0,Y 474.319,Z 384.457,A -85,B 0,C 180,E1 20520.242,E2 20520.242} C_VEL
LIN {X 0,Y 477.325,Z 385.997,A -85,B 0,C 180,E1 20516.096,E2 20516.096} C_VEL
LIN {X 0,Y 479.237,Z 389.811,A -85,B 0,C 180,E1 20514.132,E2 20514.132} C_VEL
LIN {X 0,Y 483.103,Z 392.764,A -85,B 0,C 180,E1 20511.43,E2 20511.43} C_VEL
LIN {X 0,Y 485.38,Z 396.457,A -85,B 0,C 180,E1 20509.975,E2 20509.975} C_VEL
LIN {X 0,Y 488.665,Z 399.141,A -85,B 0,C 180,E1 20508.283,E2 20508.283} C_VEL
LIN {X 0,Y 491.74,Z 403.433,A -85,B 0,C 180,E1 20506.776,E2 20506.776} C_VEL
LIN {X 0,Y 494.029,Z 405.581,A -85,B 0,C 180,E1 20505.794,E2 20505.794} C_VEL
LIN {X 0,Y 497.328,Z 409.833,A -85,B 0,C 180,E1 20504.431,E2 20504.431} C_VEL
LIN {X 0,Y 499.229,Z 411.749,A -85,B 0,C 180,E1 20503.716,E2 20503.716} C_VEL
LIN {X 0,Y 502.988,Z 416.29,A -85,B 0,C 180,E1 20502.353,E2 20502.353} C_VEL
LIN {X 0,Y 509.23,Z 424.032,A -85,B 0,C 180,E1 20500.291,E2 20500.291} C_VEL
LIN {X 0,Y 514.109,Z 430.092,A -85,B 0,C 180,E1 20498.822,E2 20498.822} C_VEL
LIN {X 0,Y 520.495,Z 438.148,A -85,B 0,C 180,E1 20497.047,E2 20497.047} C_VEL
LIN {X 0,Y 530.107,Z 451.92,A -85,B 0,C 180,E1 20494.589,E2 20494.589} C_VEL
LIN {X 0,Y 539.235,Z 465.634,A -85,B 0,C 180,E1 20492.472,E2 20492.472} C_VEL
LIN {X 0,Y 550.499,Z 483.186,A -85,B 0,C 180,E1 20490.093,E2 20490.093} C_VEL
LIN {X 0,Y 540.02,Z 690.839,A -85,B 0,C 180,E1 20486.925,E2 20486.925} C_VEL
LIN {X 0,Y 533.319,Z 825.583,A -85,B 0,C 180,E1 20484.868,E2 20484.868} C_VEL
LIN {X 0,Y 530.911,Z 852.353,A -85,B 0,C 180,E1 20484.36,E2 20484.36} C_VEL
LIN {X 0,Y 527.438,Z 879.241,A -85,B 0,C 180,E1 20483.663,E2 20483.663} C_VEL
LIN {X 0,Y 524.124,Z 900.561,A -85,B 0,C 180,E1 20482.974,E2 20482.974} C_VEL
LIN {X 0,Y 520.521,Z 920.846,A -85,B 0,C 180,E1 20482.189,E2 20482.189} C_VEL
LIN {X 0,Y 516.243,Z 942.2,A -85,B 0,C 180,E1 20481.22,E2 20481.22} C_VEL
LIN {X 0,Y 510.661,Z 967.367,A -85,B 0,C 180,E1 20479.87,E2 20479.87} C_VEL
LIN {X 0,Y 504.847,Z 990.525,A -85,B 0,C 180,E1 20478.386,E2 20478.386} C_VEL
LIN {X 0,Y 499.97,Z 1008.75,A -85,B 0,C 180,E1 20477.049,E2 20477.049} C_VEL
LIN {X 0,Y 495.119,Z 1025.907,A -85,B 0,C 180,E1 20475.633,E2 20475.633} C_VEL
LIN {X 0,Y 489.977,Z 1043.351,A -85,B 0,C 180,E1 20474.014,E2 20474.014} C_VEL
LIN {X 0,Y 483.838,Z 1063.664,A -85,B 0,C 180,E1 20471.873,E2 20471.873} C_VEL
LIN {X 0,Y 477.754,Z 1082.943,A -85,B 0,C 180,E1 20469.51,E2 20469.51} C_VEL
LIN {X 0,Y 472.798,Z 1098.61,A -85,B 0,C 180,E1 20467.328,E2 20467.328} C_VEL
LIN {X 0,Y 468.45,Z 1112.446,A -85,B 0,C 180,E1 20465.164,E2 20465.164} C_VEL
LIN {X 0,Y 464.17,Z 1126.313,A -85,B 0,C 180,E1 20462.729,E2 20462.729} C_VEL
LIN {X 0,Y 459.456,Z 1142.454,A -85,B 0,C 180,E1 20459.46,E2 20459.46} C_VEL
LIN {X 0,Y 456.22,Z 1154.176,A -85,B 0,C 180,E1 20456.697,E2 20456.697} C_VEL
LIN {X 0,Y 453.763,Z 1164.035,A -85,B 0,C 180,E1 20454.057,E2 20454.057} C_VEL
LIN {X 0,Y 451.841,Z 1172.696,A -85,B 0,C 180,E1 20451.415,E2 20451.415} C_VEL
LIN {X 0,Y 450.261,Z 1180.936,A -85,B 0,C 180,E1 20448.515,E2 20448.515} C_VEL
LIN {X 0,Y 448.971,Z 1189.53,A -85,B 0,C 180,E1 20444.839,E2 20444.839} C_VEL
LIN {X 0,Y 448.359,Z 1195.066,A -85,B 0,C 180,E1 20441.839,E2 20441.839} C_VEL
LIN {X 0,Y 448.088,Z 1198.861,A -85,B 0,C 180,E1 20439.245,E2 20439.245} C_VEL
LIN {X 0,Y 447.962,Z 1201.73,A -85,B 0,C 180,E1 20436.644,E2 20436.644} C_VEL
LIN {X 0,Y 447.916,Z 1203.631,A -85,B 0,C 180,E1 20434.096,E2 20434.096} C_VEL
LIN {X 0,Y 447.91,Z 1204.635,A -85,B 0,C 180,E1 20431.535,E2 20431.535} C_VEL
LIN {X 0,Y 447.909,Z 1204.726,A -85,B 0,C 180,E1 20428.977,E2 20428.977} C_VEL
LIN {X 0,Y 447.914,Z 1203.904,A -85,B 0,C 180,E1 20426.416,E2 20426.416} C_VEL
LIN {X 0,Y 447.949,Z 1202.166,A -85,B 0,C 180,E1 20423.85,E2 20423.85} C_VEL
LIN {X 0,Y 448.056,Z 1199.502,A -85,B 0,C 180,E1 20421.272,E2 20421.272} C_VEL
LIN {X 0,Y 448.281,Z 1195.894,A -85,B 0,C 180,E1 20418.681,E2 20418.681} C_VEL
LIN {X 0,Y 448.783,Z 1191.061,A -85,B 0,C 180,E1 20415.946,E2 20415.946} C_VEL
LIN {X 0,Y 449.515,Z 1185.436,A -85,B 0,C 180,E1 20413.325,E2 20413.325} C_VEL
LIN {X 0,Y 450.728,Z 1178.331,A -85,B 0,C 180,E1 20410.531,E2 20410.531} C_VEL
LIN {X 0,Y 452.744,Z 1168.584,A -85,B 0,C 180,E1 20407.265,E2 20407.265} C_VEL
LIN {X 0,Y 455.56,Z 1156.736,A -85,B 0,C 180,E1 20403.963,E2 20403.963} C_VEL
LIN {X 0,Y 458.437,Z 1145.901,A -85,B 0,C 180,E1 20401.326,E2 20401.326} C_VEL
LIN {X 0,Y 461.988,Z 1133.747,A -85,B 0,C 180,E1 20398.707,E2 20398.707} C_VEL
LIN {X 0,Y 466.885,Z 1118.06,A -85,B 0,C 180,E1 20395.721,E2 20395.721} C_VEL
LIN {X 0,Y 472.423,Z 1100.748,A -85,B 0,C 180,E1 20392.902,E2 20392.902} C_VEL
LIN {X 0,Y 477.462,Z 1085.419,A -85,B 0,C 180,E1 20390.694,E2 20390.694} C_VEL
LIN {X 0,Y 482.932,Z 1068.891,A -85,B 0,C 180,E1 20388.579,E2 20388.579} C_VEL
LIN {X 0,Y 490.03,Z 1047.179,A -85,B 0,C 180,E1 20386.155,E2 20386.155} C_VEL
LIN {X 0,Y 496.237,Z 1027.347,A -85,B 0,C 180,E1 20384.251,E2 20384.251} C_VEL
LIN {X 0,Y 501.656,Z 1009.453,A -85,B 0,C 180,E1 20382.738,E2 20382.738} C_VEL
LIN {X 0,Y 506.698,Z 991.92,A -85,B 0,C 180,E1 20381.423,E2 20381.423} C_VEL
LIN {X 0,Y 511.999,Z 972.329,A -85,B 0,C 180,E1 20380.126,E2 20380.126} C_VEL
LIN {X 0,Y 518.293,Z 947.2,A -85,B 0,C 180,E1 20378.7,E2 20378.7} C_VEL
LIN {X 0,Y 523.535,Z 923.179,A -85,B 0,C 180,E1 20377.573,E2 20377.573} C_VEL
LIN {X 0,Y 527.552,Z 902.574,A -85,B 0,C 180,E1 20376.757,E2 20376.757} C_VEL
LIN {X 0,Y 531.156,Z 881.438,A -85,B 0,C 180,E1 20376.056,E2 20376.056} C_VEL
LIN {X 0,Y 534.276,Z 859.784,A -85,B 0,C 180,E1 20375.468,E2 20375.468} C_VEL
LIN {X 0,Y 537.415,Z 832.393,A -85,B 0,C 180,E1 20374.894,E2 20374.894} C_VEL
LIN {X 0,Y 540.233,Z 787.042,A -85,B 0,C 180,E1 20374.169,E2 20374.169} C_VEL
LIN {X 0,Y 552.91,Z 564.716,A -85,B 0,C 180,E1 20370.733,E2 20370.733} C_VEL
LIN {X 0,Y 557.673,Z 485.041,A -85,B 0,C 180,E1 20369.489,E2 20369.489} C_VEL
LIN {X 0,Y 547.892,Z 469.501,A -85,B 0,C 180,E1 20366.91,E2 20366.91} C_VEL
LIN {X 0,Y 538.886,Z 456.3,A -85,B 0,C 180,E1 20364.209,E2 20364.209} C_VEL
LIN {X 0,Y 533.17,Z 448.271,A -85,B 0,C 180,E1 20362.261,E2 20362.261} C_VEL
LIN {X 0,Y 529.003,Z 442.931,A -85,B 0,C 180,E1 20360.699,E2 20360.699} C_VEL
LIN {X 0,Y 524.948,Z 437.779,A -85,B 0,C 180,E1 20359.009,E2 20359.009} C_VEL
LIN {X 0,Y 521.408,Z 433.366,A -85,B 0,C 180,E1 20357.35,E2 20357.35} C_VEL
LIN {X 0,Y 520.46,Z 432.108,A -85,B 0,C 180,E1 20356.864,E2 20356.864} C_VEL
LIN {X 0,Y 517.028,Z 428.277,A -85,B 0,C 180,E1 20354.962,E2 20354.962} C_VEL
LIN {X 0,Y 515.947,Z 426.466,A -85,B 0,C 180,E1 20354.248,E2 20354.248} C_VEL
LIN {X 0,Y 512.562,Z 423.231,A -85,B 0,C 180,E1 20351.82,E2 20351.82} C_VEL
LIN {X 0,Y 511.015,Z 420.246,A -85,B 0,C 180,E1 20350.257,E2 20350.257} C_VEL
LIN {X 0,Y 507.64,Z 417.789,A -85,B 0,C 180,E1 20344.292,E2 20344.292} C_VEL
LIN {X 0,Y 507.916,Z 418.073,A -85,B 0,C 180,E1 20341.241,E2 20341.241} C_VEL
LIN {X 0,Y 511.247,Z 420.515,A -85,B 0,C 180,E1 20336.299,E2 20336.299} C_VEL
LIN {X 0,Y 513.239,Z 424.151,A -85,B 0,C 180,E1 20334.41,E2 20334.41} C_VEL
LIN {X 0,Y 516.294,Z 426.923,A -85,B 0,C 180,E1 20332.321,E2 20332.321} C_VEL
LIN {X 0,Y 519.192,Z 431.017,A -85,B 0,C 180,E1 20330.578,E2 20330.578} C_VEL
LIN {X 0,Y 521.204,Z 432.967,A -85,B 0,C 180,E1 20329.555,E2 20329.555} C_VEL
LIN {X 0,Y 524.684,Z 437.51,A -85,B 0,C 180,E1 20327.899,E2 20327.899} C_VEL
LIN {X 0,Y 526.147,Z 439.295,A -85,B 0,C 180,E1 20327.265,E2 20327.265} C_VEL
LIN {X 0,Y 530.724,Z 445.104,A -85,B 0,C 180,E1 20325.433,E2 20325.433} C_VEL
LIN {X 0,Y 535.316,Z 451.032,A -85,B 0,C 180,E1 20323.785,E2 20323.785} C_VEL
LIN {X 0,Y 539.647,Z 456.721,A -85,B 0,C 180,E1 20322.365,E2 20322.365} C_VEL
LIN {X 0,Y 545.719,Z 464.809,A -85,B 0,C 180,E1 20320.548,E2 20320.548} C_VEL
LIN {X 0,Y 554.273,Z 476.995,A -85,B 0,C 180,E1 20318.24,E2 20318.24} C_VEL
LIN {X 0,Y 557.699,Z 482.725,A -85,B 0,C 180,E1 20317.365,E2 20317.365} C_VEL
LIN {X 0,Y 544.783,Z 702.167,A -85,B 0,C 180,E1 20313.967,E2 20313.967} C_VEL
LIN {X 0,Y 538.063,Z 819.34,A -85,B 0,C 180,E1 20312.143,E2 20312.143} C_VEL
LIN {X 0,Y 535.373,Z 846.737,A -85,B 0,C 180,E1 20311.612,E2 20311.612} C_VEL
LIN {X 0,Y 531.677,Z 873.076,A -85,B 0,C 180,E1 20310.912,E2 20310.912} C_VEL
LIN {X 0,Y 528.176,Z 893.993,A -85,B 0,C 180,E1 20310.222,E2 20310.222} C_VEL
LIN {X 0,Y 524.31,Z 914.128,A -85,B 0,C 180,E1 20309.43,E2 20309.43} C_VEL
LIN {X 0,Y 519.704,Z 935.444,A -85,B 0,C 180,E1 20308.445,E2 20308.445} C_VEL
LIN {X 0,Y 513.735,Z 960.316,A -85,B 0,C 180,E1 20307.085,E2 20307.085} C_VEL
LIN {X 0,Y 507.637,Z 982.819,A -85,B 0,C 180,E1 20305.616,E2 20305.616} C_VEL
LIN {X 0,Y 502.477,Z 1000.739,A -85,B 0,C 180,E1 20304.278,E2 20304.278} C_VEL
LIN {X 0,Y 497.121,Z 1018.347,A -85,B 0,C 180,E1 20302.794,E2 20302.794} C_VEL
LIN {X 0,Y 491.461,Z 1036.214,A -85,B 0,C 180,E1 20301.094,E2 20301.094} C_VEL
LIN {X 0,Y 484.745,Z 1056.963,A -85,B 0,C 180,E1 20298.839,E2 20298.839} C_VEL
LIN {X 0,Y 478.443,Z 1075.565,A -85,B 0,C 180,E1 20296.482,E2 20296.482} C_VEL
LIN {X 0,Y 473.446,Z 1090.457,A -85,B 0,C 180,E1 20294.349,E2 20294.349} C_VEL
LIN {X 0,Y 468.745,Z 1104.641,A -85,B 0,C 180,E1 20292.07,E2 20292.07} C_VEL
LIN {X 0,Y 463.871,Z 1119.91,A -85,B 0,C 180,E1 20289.3,E2 20289.3} C_VEL
LIN {X 0,Y 459.276,Z 1134.932,A -85,B 0,C 180,E1 20286.127,E2 20286.127} C_VEL
LIN {X 0,Y 456.245,Z 1145.731,A -85,B 0,C 180,E1 20283.522,E2 20283.522} C_VEL
LIN {X 0,Y 453.785,Z 1155.38,A -85,B 0,C 180,E1 20280.89,E2 20280.89} C_VEL
LIN {X 0,Y 452.142,Z 1162.468,A -85,B 0,C 180,E1 20278.708,E2 20278.708} C_VEL
LIN {X 0,Y 450.568,Z 1165.345,A -85,B 0,C 180,E1 20277.812,E2 20277.812} C_VEL
LIN {X 0,Y 443.074,Z 1172.589,A -85,B 0,C 180,E1 20275.436,E2 20275.436} C_VEL
LIN {X 0,Y 441.98,Z 1174.583,A -85,B 0,C 180,E1 20274.623,E2 20274.623} C_VEL
LIN {X 0,Y 440.91,Z 1181.378,A -85,B 0,C 180,E1 20271.414,E2 20271.414} C_VEL
LIN {X 0,Y 440.344,Z 1186.311,A -85,B 0,C 180,E1 20268.535,E2 20268.535} C_VEL
LIN {X 0,Y 440.068,Z 1190.101,A -85,B 0,C 180,E1 20265.687,E2 20265.687} C_VEL
LIN {X 0,Y 439.945,Z 1193.035,A -85,B 0,C 180,E1 20262.602,E2 20262.602} C_VEL
LIN {X 0,Y 439.913,Z 1194.823,A -85,B 0,C 180,E1 20259.155,E2 20259.155} C_VEL
LIN {X 0,Y 439.916,Z 1195.056,A -85,B 0,C 180,E1 20256.132,E2 20256.132} C_VEL
LIN {X 0,Y 439.914,Z 1194.258,A -85,B 0,C 180,E1 20253.388,E2 20253.388} C_VEL
LIN {X 0,Y 439.961,Z 1192.484,A -85,B 0,C 180,E1 20250.651,E2 20250.651} C_VEL
LIN {X 0,Y 440.099,Z 1189.585,A -85,B 0,C 180,E1 20247.787,E2 20247.787} C_VEL
LIN {X 0,Y 440.44,Z 1185.398,A -85,B 0,C 180,E1 20244.79,E2 20244.79} C_VEL
LIN {X 0,Y 441.261,Z 1178.983,A -85,B 0,C 180,E1 20241.268,E2 20241.268} C_VEL
LIN {X 0,Y 442.613,Z 1171.075,A -85,B 0,C 180,E1 20237.873,E2 20237.873} C_VEL
LIN {X 0,Y 444.292,Z 1163.108,A -85,B 0,C 180,E1 20235.001,E2 20235.001} C_VEL
LIN {X 0,Y 446.443,Z 1154.337,A -85,B 0,C 180,E1 20232.267,E2 20232.267} C_VEL
LIN {X 0,Y 449.322,Z 1143.86,A -85,B 0,C 180,E1 20229.415,E2 20229.415} C_VEL
LIN {X 0,Y 453.774,Z 1128.922,A -85,B 0,C 180,E1 20225.944,E2 20225.944} C_VEL
LIN {X 0,Y 457.822,Z 1116.231,A -85,B 0,C 180,E1 20223.403,E2 20223.403} C_VEL
LIN {X 0,Y 461.983,Z 1103.524,A -85,B 0,C 180,E1 20221.143,E2 20221.143} C_VEL
LIN {X 0,Y 466.667,Z 1089.446,A -85,B 0,C 180,E1 20218.912,E2 20218.912} C_VEL
LIN {X 0,Y 472.81,Z 1071.16,A -85,B 0,C 180,E1 20216.355,E2 20216.355} C_VEL
LIN {X 0,Y 479.27,Z 1051.149,A -85,B 0,C 180,E1 20213.963,E2 20213.963} C_VEL
LIN {X 0,Y 484.585,Z 1034.426,A -85,B 0,C 180,E1 20212.207,E2 20212.207} C_VEL
LIN {X 0,Y 489.88,Z 1017.165,A -85,B 0,C 180,E1 20210.598,E2 20210.598} C_VEL
LIN {X 0,Y 495.287,Z 998.694,A -85,B 0,C 180,E1 20209.074,E2 20209.074} C_VEL
LIN {X 0,Y 501.839,Z 974.709,A -85,B 0,C 180,E1 20207.358,E2 20207.358} C_VEL
LIN {X 0,Y 507.402,Z 952.137,A -85,B 0,C 180,E1 20205.995,E2 20205.995} C_VEL
LIN {X 0,Y 511.716,Z 932.873,A -85,B 0,C 180,E1 20204.983,E2 20204.983} C_VEL
LIN {X 0,Y 515.793,Z 912.932,A -85,B 0,C 180,E1 20204.081,E2 20204.081} C_VEL
LIN {X 0,Y 519.536,Z 892.242,A -85,B 0,C 180,E1 20203.281,E2 20203.281} C_VEL
LIN {X 0,Y 523.547,Z 866.598,A -85,B 0,C 180,E1 20202.464,E2 20202.464} C_VEL
LIN {X 0,Y 526.748,Z 839.766,A -85,B 0,C 180,E1 20201.813,E2 20201.813} C_VEL
LIN {X 0,Y 528.75,Z 817.021,A -85,B 0,C 180,E1 20201.391,E2 20201.391} C_VEL
LIN {X 0,Y 539.244,Z 612.8,A -85,B 0,C 180,E1 20198.267,E2 20198.267} C_VEL
LIN {X 0,Y 545.981,Z 484.659,A -85,B 0,C 180,E1 20196.295,E2 20196.295} C_VEL
LIN {X 0,Y 538.466,Z 473.296,A -85,B 0,C 180,E1 20194.691,E2 20194.691} C_VEL
LIN {X 0,Y 528.524,Z 459.285,A -85,B 0,C 180,E1 20192.403,E2 20192.403} C_VEL
LIN {X 0,Y 518.311,Z 445.463,A -85,B 0,C 180,E1 20189.786,E2 20189.786} C_VEL
LIN {X 0,Y 509.75,Z 434.534,A -85,B 0,C 180,E1 20187.323,E2 20187.323} C_VEL
LIN {X 0,Y 505.19,Z 428.842,A -85,B 0,C 180,E1 20185.876,E2 20185.876} C_VEL
LIN {X 0,Y 501.06,Z 423.709,A -85,B 0,C 180,E1 20184.461,E2 20184.461} C_VEL
LIN {X 0,Y 497.205,Z 418.855,A -85,B 0,C 180,E1 20183.026,E2 20183.026} C_VEL
LIN {X 0,Y 493.158,Z 414.346,A -85,B 0,C 180,E1 20181.405,E2 20181.405} C_VEL
LIN {X 0,Y 491.895,Z 412.448,A -85,B 0,C 180,E1 20180.838,E2 20180.838} C_VEL
LIN {X 0,Y 488.293,Z 408.714,A -85,B 0,C 180,E1 20179.188,E2 20179.188} C_VEL
LIN {X 0,Y 486.723,Z 406.384,A -85,B 0,C 180,E1 20178.365,E2 20178.365} C_VEL
LIN {X 0,Y 483.431,Z 403.481,A -85,B 0,C 180,E1 20176.585,E2 20176.585} C_VEL
LIN {X 0,Y 481.505,Z 400.181,A -85,B 0,C 180,E1 20175.291,E2 20175.291} C_VEL
LIN {X 0,Y 478.051,Z 397.586,A -85,B 0,C 180,E1 20172.81,E2 20172.81} C_VEL
LIN {X 0,Y 476.004,Z 393.662,A -85,B 0,C 180,E1 20170.653,E2 20170.653} C_VEL
LIN {X 0,Y 472.671,Z 391.847,A -85,B 0,C 180,E1 20164.125,E2 20164.125} C_VEL
LIN {X 0,Y 473.392,Z 392.447,A -85,B 0,C 180,E1 20160.121,E2 20160.121} C_VEL
LIN {X 0,Y 476.218,Z 393.97,A -85,B 0,C 180,E1 20156.208,E2 20156.208} C_VEL
LIN {X 0,Y 478.252,Z 397.852,A -85,B 0,C 180,E1 20154.12,E2 20154.12} C_VEL
LIN {X 0,Y 481.753,Z 400.483,A -85,B 0,C 180,E1 20151.646,E2 20151.646} C_VEL
LIN {X 0,Y 484.129,Z 404.287,A -85,B 0,C 180,E1 20150.107,E2 20150.107} C_VEL
LIN {X 0,Y 487.165,Z 406.778,A -85,B 0,C 180,E1 20148.516,E2 20148.516} C_VEL
LIN {X 0,Y 490.256,Z 411.107,A -85,B 0,C 180,E1 20146.975,E2 20146.975} C_VEL
LIN {X 0,Y 492.384,Z 413.135,A -85,B 0,C 180,E1 20146.046,E2 20146.046} C_VEL
LIN {X 0,Y 495.777,Z 417.507,A -85,B 0,C 180,E1 20144.62,E2 20144.62} C_VEL
LIN {X 0,Y 497.576,Z 419.42,A -85,B 0,C 180,E1 20143.93,E2 20143.93} C_VEL
LIN {X 0,Y 501.54,Z 424.108,A -85,B 0,C 180,E1 20142.48,E2 20142.48} C_VEL
LIN {X 0,Y 507.552,Z 431.844,A -85,B 0,C 180,E1 20140.463,E2 20140.463} C_VEL
LIN {X 0,Y 512.128,Z 437.564,A -85,B 0,C 180,E1 20139.066,E2 20139.066} C_VEL
LIN {X 0,Y 518.351,Z 445.537,A -85,B 0,C 180,E1 20137.307,E2 20137.307} C_VEL
LIN {X 0,Y 527.759,Z 459.239,A -85,B 0,C 180,E1 20134.858,E2 20134.858} C_VEL
LIN {X 0,Y 536.475,Z 472.503,A -85,B 0,C 180,E1 20132.8,E2 20132.8} C_VEL
LIN {X 0,Y 545.993,Z 487.46,A -85,B 0,C 180,E1 20130.739,E2 20130.739} C_VEL
LIN {X 0,Y 535.126,Z 696.119,A -85,B 0,C 180,E1 20127.543,E2 20127.543} C_VEL
LIN {X 0,Y 528.463,Z 825.634,A -85,B 0,C 180,E1 20125.557,E2 20125.557} C_VEL
LIN {X 0,Y 525.946,Z 852.877,A -85,B 0,C 180,E1 20125.038,E2 20125.038} C_VEL
LIN {X 0,Y 522.398,Z 879.463,A -85,B 0,C 180,E1 20124.345,E2 20124.345} C_VEL
LIN {X 0,Y 518.946,Z 901.018,A -85,B 0,C 180,E1 20123.645,E2 20123.645} C_VEL
LIN {X 0,Y 515.225,Z 921.346,A -85,B 0,C 180,E1 20122.855,E2 20122.855} C_VEL
LIN {X 0,Y 510.85,Z 942.55,A -85,B 0,C 180,E1 20121.888,E2 20121.888} C_VEL
LIN {X 0,Y 504.866,Z 968.56,A -85,B 0,C 180,E1 20120.478,E2 20120.478} C_VEL
LIN {X 0,Y 499.124,Z 990.768,A -85,B 0,C 180,E1 20119.044,E2 20119.044} C_VEL
LIN {X 0,Y 494.092,Z 1008.983,A -85,B 0,C 180,E1 20117.7,E2 20117.7} C_VEL
LIN {X 0,Y 488.882,Z 1026.797,A -85,B 0,C 180,E1 20116.216,E2 20116.216} C_VEL
LIN {X 0,Y 483.027,Z 1046.024,A -85,B 0,C 180,E1 20114.399,E2 20114.399} C_VEL
LIN {X 0,Y 475.923,Z 1068.361,A -85,B 0,C 180,E1 20111.949,E2 20111.949} C_VEL
LIN {X 0,Y 470.483,Z 1084.989,A -85,B 0,C 180,E1 20109.847,E2 20109.847} C_VEL
LIN {X 0,Y 465.62,Z 1099.83,A -85,B 0,C 180,E1 20107.734,E2 20107.734} C_VEL
LIN {X 0,Y 460.858,Z 1114.426,A -85,B 0,C 180,E1 20105.399,E2 20105.399} C_VEL
LIN {X 0,Y 455.411,Z 1131.587,A -85,B 0,C 180,E1 20102.243,E2 20102.243} C_VEL
LIN {X 0,Y 451.43,Z 1144.63,A -85,B 0,C 180,E1 20099.452,E2 20099.452} C_VEL
LIN {X 0,Y 448.427,Z 1155.207,A -85,B 0,C 180,E1 20096.885,E2 20096.885} C_VEL
LIN {X 0,Y 445.917,Z 1164.866,A -85,B 0,C 180,E1 20094.226,E2 20094.226} C_VEL
LIN {X 0,Y 443.6,Z 1175.054,A -85,B 0,C 180,E1 20091.001,E2 20091.001} C_VEL
LIN {X 0,Y 441.851,Z 1184.138,A -85,B 0,C 180,E1 20087.515,E2 20087.515} C_VEL
LIN {X 0,Y 440.91,Z 1190.467,A -85,B 0,C 180,E1 20084.579,E2 20084.579} C_VEL
LIN {X 0,Y 440.352,Z 1195.394,A -85,B 0,C 180,E1 20081.792,E2 20081.792} C_VEL
LIN {X 0,Y 440.082,Z 1199.096,A -85,B 0,C 180,E1 20079.151,E2 20079.151} C_VEL
LIN {X 0,Y 439.96,Z 1201.853,A -85,B 0,C 180,E1 20076.525,E2 20076.525} C_VEL
LIN {X 0,Y 439.914,Z 1203.682,A -85,B 0,C 180,E1 20073.91,E2 20073.91} C_VEL
LIN {X 0,Y 439.914,Z 1204.594,A -85,B 0,C 180,E1 20071.302,E2 20071.302} C_VEL
LIN {X 0,Y 439.914,Z 1204.593,A -85,B 0,C 180,E1 20068.698,E2 20068.698} C_VEL
LIN {X 0,Y 439.914,Z 1203.679,A -85,B 0,C 180,E1 20066.09,E2 20066.09} C_VEL
LIN {X 0,Y 439.96,Z 1201.847,A -85,B 0,C 180,E1 20063.475,E2 20063.475} C_VEL
LIN {X 0,Y 440.082,Z 1199.088,A -85,B 0,C 180,E1 20060.849,E2 20060.849} C_VEL
LIN {X 0,Y 440.352,Z 1195.384,A -85,B 0,C 180,E1 20058.208,E2 20058.208} C_VEL
LIN {X 0,Y 440.909,Z 1190.453,A -85,B 0,C 180,E1 20055.421,E2 20055.421} C_VEL
LIN {X 0,Y 441.849,Z 1184.116,A -85,B 0,C 180,E1 20052.484,E2 20052.484} C_VEL
LIN {X 0,Y 443.677,Z 1174.615,A -85,B 0,C 180,E1 20048.865,E2 20048.865} C_VEL
LIN {X 0,Y 445.913,Z 1164.833,A -85,B 0,C 180,E1 20045.774,E2 20045.774} C_VEL
LIN {X 0,Y 448.454,Z 1155.103,A -85,B 0,C 180,E1 20043.089,E2 20043.089} C_VEL
LIN {X 0,Y 451.62,Z 1144.135,A -85,B 0,C 180,E1 20040.416,E2 20040.416} C_VEL
LIN {X 0,Y 456.286,Z 1129.281,A -85,B 0,C 180,E1 20037.231,E2 20037.231} C_VEL
LIN {X 0,Y 461.479,Z 1113.482,A -85,B 0,C 180,E1 20034.343,E2 20034.343} C_VEL
LIN {X 0,Y 466.355,Z 1099.162,A -85,B 0,C 180,E1 20032.025,E2 20032.025} C_VEL
LIN {X 0,Y 471.518,Z 1084.172,A -85,B 0,C 180,E1 20029.862,E2 20029.862} C_VEL
LIN {X 0,Y 477.698,Z 1066.342,A -85,B 0,C 180,E1 20027.583,E2 20027.583} C_VEL
LIN {X 0,Y 485.046,Z 1044.422,A -85,B 0,C 180,E1 20025.172,E2 20025.172} C_VEL
LIN {X 0,Y 490.94,Z 1026.329,A -85,B 0,C 180,E1 20023.444,E2 20023.444} C_VEL
LIN {X 0,Y 496.556,Z 1008.427,A -85,B 0,C 180,E1 20021.934,E2 20021.934} C_VEL
LIN {X 0,Y 502.059,Z 989.938,A -85,B 0,C 180,E1 20020.557,E2 20020.557} C_VEL
LIN {X 0,Y 508.299,Z 967.565,A -85,B 0,C 180,E1 20019.104,E2 20019.104} C_VEL
LIN {X 0,Y 514.533,Z 942.397,A -85,B 0,C 180,E1 20017.731,E2 20017.731} C_VEL
LIN {X 0,Y 519.227,Z 921.404,A -85,B 0,C 180,E1 20016.767,E2 20016.767} C_VEL
LIN {X 0,Y 523.242,Z 901.197,A -85,B 0,C 180,E1 20015.976,E2 20015.976} C_VEL
LIN {X 0,Y 526.967,Z 879.833,A -85,B 0,C 180,E1 20015.279,E2 20015.279} C_VEL
LIN {X 0,Y 530.498,Z 855.631,A -85,B 0,C 180,E1 20014.639,E2 20014.639} C_VEL
LIN {X 0,Y 533.551,Z 826.902,A -85,B 0,C 180,E1 20014.073,E2 20014.073} C_VEL
LIN {X 0,Y 538.001,Z 752.764,A -85,B 0,C 180,E1 20012.909,E2 20012.909} C_VEL
LIN {X 0,Y 551.124,Z 532.852,A -85,B 0,C 180,E1 20009.499,E2 20009.499} C_VEL
LIN {X 0,Y 553.784,Z 489.792,A -85,B 0,C 180,E1 20008.822,E2 20008.822} C_VEL
LIN {X 0,Y 545.069,Z 475.743,A -85,B 0,C 180,E1 20006.443,E2 20006.443} C_VEL
LIN {X 0,Y 536.569,Z 463.15,A -85,B 0,C 180,E1 20003.82,E2 20003.82} C_VEL
LIN {X 0,Y 531.338,Z 455.664,A -85,B 0,C 180,E1 20001.993,E2 20001.993} C_VEL
LIN {X 0,Y 527.237,Z 450.351,A -85,B 0,C 180,E1 20000.423,E2 20000.423} C_VEL
LIN {X 0,Y 523.379,Z 445.37,A -85,B 0,C 180,E1 19998.779,E2 19998.779} C_VEL
LIN {X 0,Y 519.818,Z 440.776,A -85,B 0,C 180,E1 19997.067,E2 19997.067} C_VEL
LIN {X 0,Y 515.453,Z 435.55,A -85,B 0,C 180,E1 19994.606,E2 19994.606} C_VEL
LIN {X 0,Y 514.634,Z 434.251,A -85,B 0,C 180,E1 19994.056,E2 19994.056} C_VEL
LIN {X 0,Y 511.212,Z 430.751,A -85,B 0,C 180,E1 19991.508,E2 19991.508} C_VEL
LIN {X 0,Y 509.934,Z 428.155,A -85,B 0,C 180,E1 19990.164,E2 19990.164} C_VEL
LIN {X 0,Y 506.65,Z 425.714,A -85,B 0,C 180,E1 19984.188,E2 19984.188} C_VEL
LIN {X 0,Y 506.97,Z 426.074,A -85,B 0,C 180,E1 19981.13,E2 19981.13} C_VEL
LIN {X 0,Y 510.144,Z 428.46,A -85,B 0,C 180,E1 19976.404,E2 19976.404} C_VEL
LIN {X 0,Y 512.253,Z 432.188,A -85,B 0,C 180,E1 19974.399,E2 19974.399} C_VEL
LIN {X 0,Y 515.042,Z 434.763,A -85,B 0,C 180,E1 19972.47,E2 19972.47} C_VEL
LIN {X 0,Y 518.006,Z 438.901,A -85,B 0,C 180,E1 19970.669,E2 19970.669} C_VEL
LIN {X 0,Y 519.881,Z 440.847,A -85,B 0,C 180,E1 19969.696,E2 19969.696} C_VEL
LIN {X 0,Y 523.458,Z 445.413,A -85,B 0,C 180,E1 19967.983,E2 19967.983} C_VEL
LIN {X 0,Y 529.038,Z 452.635,A -85,B 0,C 180,E1 19965.665,E2 19965.665} C_VEL
LIN {X 0,Y 533.417,Z 458.365,A -85,B 0,C 180,E1 19964.061,E2 19964.061} C_VEL
LIN {X 0,Y 537.999,Z 464.485,A -85,B 0,C 180,E1 19962.533,E2 19962.533} C_VEL
LIN {X 0,Y 543.837,Z 472.432,A -85,B 0,C 180,E1 19960.757,E2 19960.757} C_VEL
LIN {X 0,Y 551.929,Z 484.126,A -85,B 0,C 180,E1 19958.534,E2 19958.534} C_VEL
LIN {X 0,Y 553.812,Z 487.512,A -85,B 0,C 180,E1 19958.033,E2 19958.033} C_VEL
LIN {X 0,Y 540.42,Z 708.03,A -85,B 0,C 180,E1 19954.611,E2 19954.611} C_VEL
LIN {X 0,Y 533.806,Z 819.529,A -85,B 0,C 180,E1 19952.87,E2 19952.87} C_VEL
LIN {X 0,Y 531.036,Z 846.936,A -85,B 0,C 180,E1 19952.338,E2 19952.338} C_VEL
LIN {X 0,Y 527.263,Z 873.108,A -85,B 0,C 180,E1 19951.643,E2 19951.643} C_VEL
LIN {X 0,Y 523.59,Z 894.395,A -85,B 0,C 180,E1 19950.942,E2 19950.942} C_VEL
LIN {X 0,Y 519.621,Z 914.486,A -85,B 0,C 180,E1 19950.15,E2 19950.15} C_VEL
LIN {X 0,Y 515.057,Z 934.981,A -85,B 0,C 180,E1 19949.205,E2 19949.205} C_VEL
LIN {X 0,Y 508.958,Z 959.762,A -85,B 0,C 180,E1 19947.855,E2 19947.855} C_VEL
LIN {X 0,Y 502.572,Z 982.608,A -85,B 0,C 180,E1 19946.366,E2 19946.366} C_VEL
LIN {X 0,Y 497.245,Z 1000.462,A -85,B 0,C 180,E1 19945.033,E2 19945.033} C_VEL
LIN {X 0,Y 491.693,Z 1018.079,A -85,B 0,C 180,E1 19943.547,E2 19943.547} C_VEL
LIN {X 0,Y 485.797,Z 1036.022,A -85,B 0,C 180,E1 19941.834,E2 19941.834} C_VEL
LIN {X 0,Y 478.813,Z 1056.795,A -85,B 0,C 180,E1 19939.565,E2 19939.565} C_VEL
LIN {X 0,Y 472.073,Z 1075.883,A -85,B 0,C 180,E1 19937.124,E2 19937.124} C_VEL
LIN {X 0,Y 466.861,Z 1090.736,A -85,B 0,C 180,E1 19934.971,E2 19934.971} C_VEL
LIN {X 0,Y 462.189,Z 1104.177,A -85,B 0,C 180,E1 19932.787,E2 19932.787} C_VEL
LIN {X 0,Y 457.549,Z 1117.827,A -85,B 0,C 180,E1 19930.299,E2 19930.299} C_VEL
LIN {X 0,Y 452.423,Z 1133.781,A -85,B 0,C 180,E1 19926.95,E2 19926.95} C_VEL
LIN {X 0,Y 448.823,Z 1145.732,A -85,B 0,C 180,E1 19924.03,E2 19924.03} C_VEL
LIN {X 0,Y 446.177,Z 1155.455,A -85,B 0,C 180,E1 19921.325,E2 19921.325} C_VEL
LIN {X 0,Y 443.944,Z 1164.734,A -85,B 0,C 180,E1 19918.373,E2 19918.373} C_VEL
LIN {X 0,Y 441.98,Z 1174.583,A -85,B 0,C 180,E1 19914.623,E2 19914.623} C_VEL
LIN {X 0,Y 440.63,Z 1176.828,A -85,B 0,C 180,E1 19913.672,E2 19913.672} C_VEL
LIN {X 0,Y 433.488,Z 1182.572,A -85,B 0,C 180,E1 19911.073,E2 19911.073} C_VEL
LIN {X 0,Y 432.663,Z 1184.015,A -85,B 0,C 180,E1 19910.294,E2 19910.294} C_VEL
LIN {X 0,Y 432.152,Z 1189.226,A -85,B 0,C 180,E1 19906.672,E2 19906.672} C_VEL
LIN {X 0,Y 431.974,Z 1192.227,A -85,B 0,C 180,E1 19903.792,E2 19903.792} C_VEL
LIN {X 0,Y 431.919,Z 1194.134,A -85,B 0,C 180,E1 19901.019,E2 19901.019} C_VEL
LIN {X 0,Y 431.915,Z 1195.045,A -85,B 0,C 180,E1 19898.386,E2 19898.386} C_VEL
LIN {X 0,Y 431.913,Z 1195.077,A -85,B 0,C 180,E1 19895.713,E2 19895.713} C_VEL
LIN {X 0,Y 431.919,Z 1194.214,A -85,B 0,C 180,E1 19893.052,E2 19893.052} C_VEL
LIN {X 0,Y 431.975,Z 1192.348,A -85,B 0,C 180,E1 19890.265,E2 19890.265} C_VEL
LIN {X 0,Y 432.139,Z 1189.348,A -85,B 0,C 180,E1 19887.348,E2 19887.348} C_VEL
LIN {X 0,Y 432.607,Z 1184.466,A -85,B 0,C 180,E1 19883.897,E2 19883.897} C_VEL
LIN {X 0,Y 433.58,Z 1177.634,A -85,B 0,C 180,E1 19880.309,E2 19880.309} C_VEL
LIN {X 0,Y 434.965,Z 1170.463,A -85,B 0,C 180,E1 19877.251,E2 19877.251} C_VEL
LIN {X 0,Y 436.69,Z 1162.791,A -85,B 0,C 180,E1 19874.462,E2 19874.462} C_VEL
LIN {X 0,Y 438.995,Z 1153.962,A -85,B 0,C 180,E1 19871.681,E2 19871.681} C_VEL
LIN {X 0,Y 442.557,Z 1141.91,A -85,B 0,C 180,E1 19868.392,E2 19868.392} C_VEL
LIN {X 0,Y 446.804,Z 1128.304,A -85,B 0,C 180,E1 19865.262,E2 19865.262} C_VEL
LIN {X 0,Y 450.904,Z 1115.993,A -85,B 0,C 180,E1 19862.777,E2 19862.777} C_VEL
LIN {X 0,Y 455.432,Z 1102.714,A -85,B 0,C 180,E1 19860.399,E2 19860.399} C_VEL
LIN {X 0,Y 460.636,Z 1087.715,A -85,B 0,C 180,E1 19858.02,E2 19858.02} C_VEL
LIN {X 0,Y 467.716,Z 1067.115,A -85,B 0,C 180,E1 19855.196,E2 19855.196} C_VEL
LIN {X 0,Y 473.476,Z 1049.989,A -85,B 0,C 180,E1 19853.166,E2 19853.166} C_VEL
LIN {X 0,Y 479.045,Z 1033.008,A -85,B 0,C 180,E1 19851.386,E2 19851.386} C_VEL
LIN {X 0,Y 485.353,Z 1012.995,A -85,B 0,C 180,E1 19849.54,E2 19849.54} C_VEL
LIN {X 0,Y 492.31,Z 989.308,A -85,B 0,C 180,E1 19847.671,E2 19847.671} C_VEL
LIN {X 0,Y 497.804,Z 969.021,A -85,B 0,C 180,E1 19846.296,E2 19846.296} C_VEL
LIN {X 0,Y 502.655,Z 949.74,A -85,B 0,C 180,E1 19845.158,E2 19845.158} C_VEL
LIN {X 0,Y 507.156,Z 930.031,A -85,B 0,C 180,E1 19844.141,E2 19844.141} C_VEL
LIN {X 0,Y 512.339,Z 904.898,A -85,B 0,C 180,E1 19843.042,E2 19843.042} C_VEL
LIN {X 0,Y 516.807,Z 878.508,A -85,B 0,C 180,E1 19842.118,E2 19842.118} C_VEL
LIN {X 0,Y 519.934,Z 856.577,A -85,B 0,C 180,E1 19841.499,E2 19841.499} C_VEL
LIN {X 0,Y 522.407,Z 835.208,A -85,B 0,C 180,E1 19841.017,E2 19841.017} C_VEL
LIN {X 0,Y 524.427,Z 810.725,A -85,B 0,C 180,E1 19840.583,E2 19840.583} C_VEL
LIN {X 0,Y 536.055,Z 590.034,A -85,B 0,C 180,E1 19837.202,E2 19837.202} C_VEL
LIN {X 0,Y 541.496,Z 489.006,A -85,B 0,C 180,E1 19835.633,E2 19835.633} C_VEL
LIN {X 0,Y 535.201,Z 479.437,A -85,B 0,C 180,E1 19834.251,E2 19834.251} C_VEL
LIN {X 0,Y 525.716,Z 465.919,A -85,B 0,C 180,E1 19832.017,E2 19832.017} C_VEL
LIN {X 0,Y 515.843,Z 452.411,A -85,B 0,C 180,E1 19829.431,E2 19829.431} C_VEL
LIN {X 0,Y 507.586,Z 441.725,A -85,B 0,C 180,E1 19827.005,E2 19827.005} C_VEL
LIN {X 0,Y 502.988,Z 435.934,A -85,B 0,C 180,E1 19825.515,E2 19825.515} C_VEL
LIN {X 0,Y 499.028,Z 430.97,A -85,B 0,C 180,E1 19824.126,E2 19824.126} C_VEL
LIN {X 0,Y 494.662,Z 425.59,A -85,B 0,C 180,E1 19822.46,E2 19822.46} C_VEL
LIN {X 0,Y 490.979,Z 421.028,A -85,B 0,C 180,E1 19820.91,E2 19820.91} C_VEL
LIN {X 0,Y 489.51,Z 419.44,A -85,B 0,C 180,E1 19820.257,E2 19820.257} C_VEL
LIN {X 0,Y 485.994,Z 415.059,A -85,B 0,C 180,E1 19818.534,E2 19818.534} C_VEL
LIN {X 0,Y 485.23,Z 414.089,A -85,B 0,C 180,E1 19818.129,E2 19818.129} C_VEL
LIN {X 0,Y 481.988,Z 411.053,A -85,B 0,C 180,E1 19816.326,E2 19816.326} C_VEL
LIN {X 0,Y 480.179,Z 407.987,A -85,B 0,C 180,E1 19815.087,E2 19815.087} C_VEL
LIN {X 0,Y 476.811,Z 405.306,A -85,B 0,C 180,E1 19812.597,E2 19812.597} C_VEL
LIN {X 0,Y 474.851,Z 401.558,A -85,B 0,C 180,E1 19810.479,E2 19810.479} C_VEL
LIN {X 0,Y 471.694,Z 399.788,A -85,B 0,C 180,E1 19804.133,E2 19804.133} C_VEL
LIN {X 0,Y 472.414,Z 400.392,A -85,B 0,C 180,E1 19800.121,E2 19800.121} C_VEL
LIN {X 0,Y 475.069,Z 401.787,A -85,B 0,C 180,E1 19796.38,E2 19796.38} C_VEL
LIN {X 0,Y 477.127,Z 405.725,A -85,B 0,C 180,E1 19794.227,E2 19794.227} C_VEL
LIN {X 0,Y 480.488,Z 408.374,A -85,B 0,C 180,E1 19791.805,E2 19791.805} C_VEL
LIN {X 0,Y 483.006,Z 412.251,A -85,B 0,C 180,E1 19790.166,E2 19790.166} C_VEL
LIN {X 0,Y 485.828,Z 414.694,A -85,B 0,C 180,E1 19788.665,E2 19788.665} C_VEL
LIN {X 0,Y 489.026,Z 419.025,A -85,B 0,C 180,E1 19787.062,E2 19787.062} C_VEL
LIN {X 0,Y 490.869,Z 420.892,A -85,B 0,C 180,E1 19786.242,E2 19786.242} C_VEL
LIN {X 0,Y 494.515,Z 425.444,A -85,B 0,C 180,E1 19784.7,E2 19784.7} C_VEL
LIN {X 0,Y 496.208,Z 427.5,A -85,B 0,C 180,E1 19784.035,E2 19784.035} C_VEL
LIN {X 0,Y 500.673,Z 432.994,A -85,B 0,C 180,E1 19782.389,E2 19782.389} C_VEL
LIN {X 0,Y 505.468,Z 439.076,A -85,B 0,C 180,E1 19780.77,E2 19780.77} C_VEL
LIN {X 0,Y 510.331,Z 445.263,A -85,B 0,C 180,E1 19779.259,E2 19779.259} C_VEL
LIN {X 0,Y 516.496,Z 453.313,A -85,B 0,C 180,E1 19777.491,E2 19777.491} C_VEL
LIN {X 0,Y 525.821,Z 467.159,A -85,B 0,C 180,E1 19775.029,E2 19775.029} C_VEL
LIN {X 0,Y 535.225,Z 481.631,A -85,B 0,C 180,E1 19772.791,E2 19772.791} C_VEL
LIN {X 0,Y 541.549,Z 491.856,A -85,B 0,C 180,E1 19771.391,E2 19771.391} C_VEL
LIN {X 0,Y 530.118,Z 704.578,A -85,B 0,C 180,E1 19768.124,E2 19768.124} C_VEL
LIN {X 0,Y 523.687,Z 825.523,A -85,B 0,C 180,E1 19766.261,E2 19766.261} C_VEL
LIN {X 0,Y 521.121,Z 852.673,A -85,B 0,C 180,E1 19765.743,E2 19765.743} C_VEL
LIN {X 0,Y 517.483,Z 879.306,A -85,B 0,C 180,E1 19765.05,E2 19765.05} C_VEL
LIN {X 0,Y 513.971,Z 900.698,A -85,B 0,C 180,E1 19764.358,E2 19764.358} C_VEL
LIN {X 0,Y 510.159,Z 921.037,A -85,B 0,C 180,E1 19763.568,E2 19763.568} C_VEL
LIN {X 0,Y 505.777,Z 941.72,A -85,B 0,C 180,E1 19762.627,E2 19762.627} C_VEL
LIN {X 0,Y 500.12,Z 966.027,A -85,B 0,C 180,E1 19761.325,E2 19761.325} C_VEL
LIN {X 0,Y 493.931,Z 989.348,A -85,B 0,C 180,E1 19759.833,E2 19759.833} C_VEL
LIN {X 0,Y 488.667,Z 1007.843,A -85,B 0,C 180,E1 19758.474,E2 19758.474} C_VEL
LIN {X 0,Y 483.297,Z 1025.665,A -85,B 0,C 180,E1 19756.993,E2 19756.993} C_VEL
LIN {X 0,Y 477.644,Z 1043.643,A -85,B 0,C 180,E1 19755.301,E2 19755.301} C_VEL
LIN {X 0,Y 470.951,Z 1064.312,A -85,B 0,C 180,E1 19753.083,E2 19753.083} C_VEL
LIN {X 0,Y 464.358,Z 1083.719,A -85,B 0,C 180,E1 19750.643,E2 19750.643} C_VEL
LIN {X 0,Y 459.261,Z 1098.678,A -85,B 0,C 180,E1 19748.51,E2 19748.51} C_VEL
LIN {X 0,Y 454.525,Z 1112.605,A -85,B 0,C 180,E1 19746.281,E2 19746.281} C_VEL
LIN {X 0,Y 449.848,Z 1126.605,A -85,B 0,C 180,E1 19743.756,E2 19743.756} C_VEL
LIN {X 0,Y 444.687,Z 1142.718,A -85,B 0,C 180,E1 19740.391,E2 19740.391} C_VEL
LIN {X 0,Y 441.222,Z 1154.164,A -85,B 0,C 180,E1 19737.615,E2 19737.615} C_VEL
LIN {X 0,Y 438.548,Z 1163.83,A -85,B 0,C 180,E1 19734.947,E2 19734.947} C_VEL
LIN {X 0,Y 436.378,Z 1172.509,A -85,B 0,C 180,E1 19732.213,E2 19732.213} C_VEL
LIN {X 0,Y 434.616,Z 1180.753,A -85,B 0,C 180,E1 19729.207,E2 19729.207} C_VEL
LIN {X 0,Y 433.136,Z 1189.35,A -85,B 0,C 180,E1 19725.395,E2 19725.395} C_VEL
LIN {X 0,Y 432.433,Z 1194.888,A -85,B 0,C 180,E1 19722.282,E2 19722.282} C_VEL
LIN {X 0,Y 432.116,Z 1198.685,A -85,B 0,C 180,E1 19719.59,E2 19719.59} C_VEL
LIN {X 0,Y 431.967,Z 1201.535,A -85,B 0,C 180,E1 19716.913,E2 19716.913} C_VEL
LIN {X 0,Y 431.918,Z 1203.457,A -85,B 0,C 180,E1 19714.248,E2 19714.248} C_VEL
LIN {X 0,Y 431.91,Z 1204.46,A -85,B 0,C 180,E1 19711.592,E2 19711.592} C_VEL
LIN {X 0,Y 431.911,Z 1204.551,A -85,B 0,C 180,E1 19708.939,E2 19708.939} C_VEL
LIN {X 0,Y 431.914,Z 1203.728,A -85,B 0,C 180,E1 19706.284,E2 19706.284} C_VEL
LIN {X 0,Y 431.956,Z 1201.988,A -85,B 0,C 180,E1 19703.621,E2 19703.621} C_VEL
LIN {X 0,Y 432.076,Z 1199.321,A -85,B 0,C 180,E1 19700.946,E2 19700.946} C_VEL
LIN {X 0,Y 432.345,Z 1195.71,A -85,B 0,C 180,E1 19698.258,E2 19698.258} C_VEL
LIN {X 0,Y 432.881,Z 1191.13,A -85,B 0,C 180,E1 19695.555,E2 19695.555} C_VEL
LIN {X 0,Y 433.711,Z 1185.552,A -85,B 0,C 180,E1 19692.837,E2 19692.837} C_VEL
LIN {X 0,Y 435.039,Z 1178.582,A -85,B 0,C 180,E1 19689.974,E2 19689.974} C_VEL
LIN {X 0,Y 437.089,Z 1169.624,A -85,B 0,C 180,E1 19686.83,E2 19686.83} C_VEL
LIN {X 0,Y 440.416,Z 1157.129,A -85,B 0,C 180,E1 19683.142,E2 19683.142} C_VEL
LIN {X 0,Y 443.791,Z 1145.849,A -85,B 0,C 180,E1 19680.287,E2 19680.287} C_VEL
LIN {X 0,Y 447.509,Z 1134.4,A -85,B 0,C 180,E1 19677.725,E2 19677.725} C_VEL
LIN {X 0,Y 451.847,Z 1121.636,A -85,B 0,C 180,E1 19675.184,E2 19675.184} C_VEL
LIN {X 0,Y 458.015,Z 1104.314,A -85,B 0,C 180,E1 19672.162,E2 19672.162} C_VEL
LIN {X 0,Y 464.178,Z 1087.084,A -85,B 0,C 180,E1 19669.582,E2 19669.582} C_VEL
LIN {X 0,Y 469.668,Z 1071.815,A -85,B 0,C 180,E1 19667.558,E2 19667.558} C_VEL
LIN {X 0,Y 475.266,Z 1056.063,A -85,B 0,C 180,E1 19665.697,E2 19665.697} C_VEL
LIN {X 0,Y 481.507,Z 1038.078,A -85,B 0,C 180,E1 19663.814,E2 19663.814} C_VEL
LIN {X 0,Y 489.35,Z 1014.519,A -85,B 0,C 180,E1 19661.686,E2 19661.686} C_VEL
LIN {X 0,Y 495.609,Z 994.359,A -85,B 0,C 180,E1 19660.128,E2 19660.128} C_VEL
LIN {X 0,Y 501.196,Z 975.157,A -85,B 0,C 180,E1 19658.829,E2 19658.829} C_VEL
LIN {X 0,Y 506.523,Z 955.459,A -85,B 0,C 180,E1 19657.669,E2 19657.669} C_VEL
LIN {X 0,Y 512.038,Z 933.164,A -85,B 0,C 180,E1 19656.54,E2 19656.54} C_VEL
LIN {X 0,Y 517.971,Z 905.506,A -85,B 0,C 180,E1 19655.389,E2 19655.389} C_VEL
LIN {X 0,Y 522.017,Z 883.375,A -85,B 0,C 180,E1 19654.643,E2 19654.643} C_VEL
LIN {X 0,Y 525.269,Z 862.38,A -85,B 0,C 180,E1 19654.063,E2 19654.063} C_VEL
LIN {X 0,Y 528.039,Z 840.479,A -85,B 0,C 180,E1 19653.582,E2 19653.582} C_VEL
LIN {X 0,Y 530.463,Z 812.673,A -85,B 0,C 180,E1 19653.095,E2 19653.095} C_VEL
LIN {X 0,Y 544.017,Z 588.346,A -85,B 0,C 180,E1 19649.612,E2 19649.612} C_VEL
LIN {X 0,Y 549.896,Z 494.452,A -85,B 0,C 180,E1 19648.125,E2 19648.125} C_VEL
LIN {X 0,Y 542.12,Z 481.721,A -85,B 0,C 180,E1 19645.921,E2 19645.921} C_VEL
LIN {X 0,Y 533.392,Z 468.705,A -85,B 0,C 180,E1 19643.124,E2 19643.124} C_VEL
LIN {X 0,Y 529.094,Z 462.549,A -85,B 0,C 180,E1 19641.566,E2 19641.566} C_VEL
LIN {X 0,Y 525.486,Z 457.767,A -85,B 0,C 180,E1 19640.146,E2 19640.146} C_VEL
LIN {X 0,Y 521.818,Z 452.958,A -85,B 0,C 180,E1 19638.547,E2 19638.547} C_VEL
LIN {X 0,Y 518.311,Z 448.311,A -85,B 0,C 180,E1 19636.82,E2 19636.82} C_VEL
LIN {X 0,Y 514.138,Z 443.256,A -85,B 0,C 180,E1 19634.414,E2 19634.414} C_VEL
LIN {X 0,Y 513.328,Z 442.03,A -85,B 0,C 180,E1 19633.862,E2 19633.862} C_VEL
LIN {X 0,Y 509.879,Z 438.261,A -85,B 0,C 180,E1 19631.195,E2 19631.195} C_VEL
LIN {X 0,Y 508.855,Z 436.062,A -85,B 0,C 180,E1 19630.072,E2 19630.072} C_VEL
LIN {X 0,Y 505.674,Z 433.656,A -85,B 0,C 180,E1 19624.196,E2 19624.196} C_VEL
LIN {X 0,Y 505.99,Z 434.022,A -85,B 0,C 180,E1 19621.132,E2 19621.132} C_VEL
LIN {X 0,Y 509,Z 436.265,A -85,B 0,C 180,E1 19616.565,E2 19616.565} C_VEL
LIN {X 0,Y 511.127,Z 440.061,A -85,B 0,C 180,E1 19614.499,E2 19614.499} C_VEL
LIN {X 0,Y 513.794,Z 442.596,A -85,B 0,C 180,E1 19612.62,E2 19612.62} C_VEL
LIN {X 0,Y 516.822,Z 446.784,A -85,B 0,C 180,E1 19610.759,E2 19610.759} C_VEL
LIN {X 0,Y 518.464,Z 448.544,A -85,B 0,C 180,E1 19609.892,E2 19609.892} C_VEL
LIN {X 0,Y 522.104,Z 453.195,A -85,B 0,C 180,E1 19608.123,E2 19608.123} C_VEL
LIN {X 0,Y 527.492,Z 460.36,A -85,B 0,C 180,E1 19605.846,E2 19605.846} C_VEL
LIN {X 0,Y 531.893,Z 466.21,A -85,B 0,C 180,E1 19604.21,E2 19604.21} C_VEL
LIN {X 0,Y 538.035,Z 474.385,A -85,B 0,C 180,E1 19602.171,E2 19602.171} C_VEL
LIN {X 0,Y 547.448,Z 487.886,A -85,B 0,C 180,E1 19599.415,E2 19599.415} C_VEL
LIN {X 0,Y 550.014,Z 492.132,A -85,B 0,C 180,E1 19598.713,E2 19598.713} C_VEL
LIN {X 0,Y 536.098,Z 714.432,A -85,B 0,C 180,E1 19595.257,E2 19595.257} C_VEL
LIN {X 0,Y 529.636,Z 819.73,A -85,B 0,C 180,E1 19593.607,E2 19593.607} C_VEL
LIN {X 0,Y 526.767,Z 847.288,A -85,B 0,C 180,E1 19593.071,E2 19593.071} C_VEL
LIN {X 0,Y 522.938,Z 873.182,A -85,B 0,C 180,E1 19592.386,E2 19592.386} C_VEL
LIN {X 0,Y 519.25,Z 894.013,A -85,B 0,C 180,E1 19591.704,E2 19591.704} C_VEL
LIN {X 0,Y 515.161,Z 914.194,A -85,B 0,C 180,E1 19590.912,E2 19590.912} C_VEL
LIN {X 0,Y 510.464,Z 934.709,A -85,B 0,C 180,E1 19589.969,E2 19589.969} C_VEL
LIN {X 0,Y 504.452,Z 958.529,A -85,B 0,C 180,E1 19588.679,E2 19588.679} C_VEL
LIN {X 0,Y 497.594,Z 982.408,A -85,B 0,C 180,E1 19587.132,E2 19587.132} C_VEL
LIN {X 0,Y 491.785,Z 1001.212,A -85,B 0,C 180,E1 19585.723,E2 19585.723} C_VEL
LIN {X 0,Y 485.854,Z 1019.365,A -85,B 0,C 180,E1 19584.177,E2 19584.177} C_VEL
LIN {X 0,Y 479.351,Z 1038.441,A -85,B 0,C 180,E1 19582.325,E2 19582.325} C_VEL
LIN {X 0,Y 471.641,Z 1060.167,A -85,B 0,C 180,E1 19579.872,E2 19579.872} C_VEL
LIN {X 0,Y 465.588,Z 1076.707,A -85,B 0,C 180,E1 19577.716,E2 19577.716} C_VEL
LIN {X 0,Y 460.335,Z 1091.036,A -85,B 0,C 180,E1 19575.61,E2 19575.61} C_VEL
LIN {X 0,Y 455.167,Z 1105.242,A -85,B 0,C 180,E1 19573.264,E2 19573.264} C_VEL
LIN {X 0,Y 449.553,Z 1121.178,A -85,B 0,C 180,E1 19570.279,E2 19570.279} C_VEL
LIN {X 0,Y 444.597,Z 1135.747,A -85,B 0,C 180,E1 19567.064,E2 19567.064} C_VEL
LIN {X 0,Y 441.213,Z 1146.524,A -85,B 0,C 180,E1 19564.352,E2 19564.352} C_VEL
LIN {X 0,Y 438.308,Z 1156.689,A -85,B 0,C 180,E1 19561.439,E2 19561.439} C_VEL
LIN {X 0,Y 435.6,Z 1167.628,A -85,B 0,C 180,E1 19557.772,E2 19557.772} C_VEL
LIN {X 0,Y 433.93,Z 1175.733,A -85,B 0,C 180,E1 19554.468,E2 19554.468} C_VEL
LIN {X 0,Y 432.955,Z 1181.721,A -85,B 0,C 180,E1 19551.542,E2 19551.542} C_VEL
LIN {X 0,Y 432.663,Z 1184.015,A -85,B 0,C 180,E1 19550.294,E2 19550.294} C_VEL
LIN {X 0,Y 431.473,Z 1185.729,A -85,B 0,C 180,E1 19549.303,E2 19549.303} C_VEL
LIN {X 0,Y 424.673,Z 1189.713,A -85,B 0,C 180,E1 19546.495,E2 19546.495} C_VEL
LIN {X 0,Y 424.081,Z 1190.583,A -85,B 0,C 180,E1 19545.755,E2 19545.755} C_VEL
LIN {X 0,Y 423.937,Z 1193.712,A -85,B 0,C 180,E1 19542.117,E2 19542.117} C_VEL
LIN {X 0,Y 423.913,Z 1195.072,A -85,B 0,C 180,E1 19538.77,E2 19538.77} C_VEL
LIN {X 0,Y 423.915,Z 1195.207,A -85,B 0,C 180,E1 19535.957,E2 19535.957} C_VEL
LIN {X 0,Y 423.919,Z 1194.362,A -85,B 0,C 180,E1 19533.11,E2 19533.11} C_VEL
LIN {X 0,Y 423.977,Z 1192.538,A -85,B 0,C 180,E1 19530.27,E2 19530.27} C_VEL
LIN {X 0,Y 424.135,Z 1189.737,A -85,B 0,C 180,E1 19527.433,E2 19527.433} C_VEL
LIN {X 0,Y 424.507,Z 1185.75,A -85,B 0,C 180,E1 19524.458,E2 19524.458} C_VEL
LIN {X 0,Y 425.346,Z 1179.929,A -85,B 0,C 180,E1 19521.075,E2 19521.075} C_VEL
LIN {X 0,Y 426.965,Z 1171.563,A -85,B 0,C 180,E1 19517.284,E2 19517.284} C_VEL
LIN {X 0,Y 428.82,Z 1163.636,A -85,B 0,C 180,E1 19514.308,E2 19514.308} C_VEL
LIN {X 0,Y 431.139,Z 1155.097,A -85,B 0,C 180,E1 19511.541,E2 19511.541} C_VEL
LIN {X 0,Y 434.058,Z 1145.406,A -85,B 0,C 180,E1 19508.798,E2 19508.798} C_VEL
LIN {X 0,Y 438.461,Z 1131.951,A -85,B 0,C 180,E1 19505.479,E2 19505.479} C_VEL
LIN {X 0,Y 443.638,Z 1116.859,A -85,B 0,C 180,E1 19502.346,E2 19502.346} C_VEL
LIN {X 0,Y 448.363,Z 1103.529,A -85,B 0,C 180,E1 19499.915,E2 19499.915} C_VEL
LIN {X 0,Y 453.51,Z 1089.231,A -85,B 0,C 180,E1 19497.606,E2 19497.606} C_VEL
LIN {X 0,Y 460.305,Z 1070.358,A -85,B 0,C 180,E1 19494.933,E2 19494.933} C_VEL
LIN {X 0,Y 466.758,Z 1051.796,A -85,B 0,C 180,E1 19492.683,E2 19492.683} C_VEL
LIN {X 0,Y 472.625,Z 1034.5,A -85,B 0,C 180,E1 19490.84,E2 19490.84} C_VEL
LIN {X 0,Y 478.477,Z 1016.557,A -85,B 0,C 180,E1 19489.151,E2 19489.151} C_VEL
LIN {X 0,Y 485.353,Z 994.414,A -85,B 0,C 180,E1 19487.331,E2 19487.331} C_VEL
LIN {X 0,Y 491.89,Z 971.137,A -85,B 0,C 180,E1 19485.715,E2 19485.715} C_VEL
LIN {X 0,Y 497.098,Z 951.114,A -85,B 0,C 180,E1 19484.518,E2 19484.518} C_VEL
LIN {X 0,Y 501.713,Z 931.541,A -85,B 0,C 180,E1 19483.497,E2 19483.497} C_VEL
LIN {X 0,Y 506.243,Z 910.314,A -85,B 0,C 180,E1 19482.55,E2 19482.55} C_VEL
LIN {X 0,Y 511.182,Z 883.606,A -85,B 0,C 180,E1 19481.561,E2 19481.561} C_VEL
LIN {X 0,Y 514.905,Z 858.48,A -85,B 0,C 180,E1 19480.831,E2 19480.831} C_VEL
LIN {X 0,Y 517.513,Z 836.856,A -85,B 0,C 180,E1 19480.335,E2 19480.335} C_VEL
LIN {X 0,Y 519.494,Z 814.335,A -85,B 0,C 180,E1 19479.927,E2 19479.927} C_VEL
LIN {X 0,Y 531.135,Z 601.065,A -85,B 0,C 180,E1 19476.644,E2 19476.644} C_VEL
LIN {X 0,Y 537.187,Z 493.458,A -85,B 0,C 180,E1 19474.981,E2 19474.981} C_VEL
LIN {X 0,Y 529.318,Z 481.617,A -85,B 0,C 180,E1 19473.185,E2 19473.185} C_VEL
LIN {X 0,Y 519.173,Z 467.317,A -85,B 0,C 180,E1 19470.657,E2 19470.657} C_VEL
LIN {X 0,Y 509.775,Z 454.491,A -85,B 0,C 180,E1 19468.019,E2 19468.019} C_VEL
LIN {X 0,Y 501.66,Z 443.972,A -85,B 0,C 180,E1 19465.438,E2 19465.438} C_VEL
LIN {X 0,Y 497.167,Z 438.376,A -85,B 0,C 180,E1 19463.844,E2 19463.844} C_VEL
LIN {X 0,Y 492.865,Z 433.027,A -85,B 0,C 180,E1 19462.169,E2 19462.169} C_VEL
LIN {X 0,Y 489.137,Z 428.205,A -85,B 0,C 180,E1 19460.554,E2 19460.554} C_VEL
LIN {X 0,Y 484.9,Z 423.333,A -85,B 0,C 180,E1 19458.515,E2 19458.515} C_VEL
LIN {X 0,Y 483.83,Z 421.835,A -85,B 0,C 180,E1 19457.934,E2 19457.934} C_VEL
LIN {X 0,Y 480.554,Z 418.624,A -85,B 0,C 180,E1 19456.065,E2 19456.065} C_VEL
LIN {X 0,Y 478.86,Z 415.785,A -85,B 0,C 180,E1 19454.882,E2 19454.882} C_VEL
LIN {X 0,Y 475.576,Z 413.024,A -85,B 0,C 180,E1 19452.384,E2 19452.384} C_VEL
LIN {X 0,Y 473.731,Z 409.461,A -85,B 0,C 180,E1 19450.335,E2 19450.335} C_VEL
LIN {X 0,Y 470.718,Z 407.728,A -85,B 0,C 180,E1 19444.142,E2 19444.142} C_VEL
LIN {X 0,Y 471.383,Z 408.293,A -85,B 0,C 180,E1 19440.243,E2 19440.243} C_VEL
LIN {X 0,Y 473.97,Z 409.734,A -85,B 0,C 180,E1 19436.493,E2 19436.493} C_VEL
LIN {X 0,Y 476.004,Z 413.598,A -85,B 0,C 180,E1 19434.334,E2 19434.334} C_VEL
LIN {X 0,Y 479.228,Z 416.249,A -85,B 0,C 180,E1 19431.964,E2 19431.964} C_VEL
LIN {X 0,Y 481.822,Z 420.143,A -85,B 0,C 180,E1 19430.263,E2 19430.263} C_VEL
LIN {X 0,Y 484.394,Z 422.41,A -85,B 0,C 180,E1 19428.872,E2 19428.872} C_VEL
LIN {X 0,Y 487.674,Z 426.82,A -85,B 0,C 180,E1 19427.207,E2 19427.207} C_VEL
LIN {X 0,Y 489.303,Z 428.533,A -85,B 0,C 180,E1 19426.468,E2 19426.468} C_VEL
LIN {X 0,Y 492.94,Z 433.088,A -85,B 0,C 180,E1 19424.905,E2 19424.905} C_VEL
LIN {X 0,Y 498.83,Z 440.446,A -85,B 0,C 180,E1 19422.652,E2 19422.652} C_VEL
LIN {X 0,Y 503.723,Z 446.756,A -85,B 0,C 180,E1 19420.972,E2 19420.972} C_VEL
LIN {X 0,Y 508.541,Z 452.952,A -85,B 0,C 180,E1 19419.453,E2 19419.453} C_VEL
LIN {X 0,Y 514.646,Z 461.087,A -85,B 0,C 180,E1 19417.677,E2 19417.677} C_VEL
LIN {X 0,Y 525.392,Z 477.312,A -85,B 0,C 180,E1 19414.827,E2 19414.827} C_VEL
LIN {X 0,Y 536.092,Z 494.433,A -85,B 0,C 180,E1 19412.297,E2 19412.297} C_VEL
LIN {X 0,Y 537.159,Z 496.4,A -85,B 0,C 180,E1 19412.053,E2 19412.053} C_VEL
LIN {X 0,Y 525.341,Z 709.714,A -85,B 0,C 180,E1 19408.767,E2 19408.767} C_VEL
LIN {X 0,Y 518.97,Z 825.676,A -85,B 0,C 180,E1 19406.972,E2 19406.972} C_VEL
LIN {X 0,Y 516.287,Z 853.218,A -85,B 0,C 180,E1 19406.445,E2 19406.445} C_VEL
LIN {X 0,Y 512.593,Z 879.465,A -85,B 0,C 180,E1 19405.759,E2 19405.759} C_VEL
LIN {X 0,Y 508.94,Z 901.102,A -85,B 0,C 180,E1 19405.057,E2 19405.057} C_VEL
LIN {X 0,Y 505.002,Z 921.51,A -85,B 0,C 180,E1 19404.261,E2 19404.261} C_VEL
LIN {X 0,Y 500.276,Z 943.179,A -85,B 0,C 180,E1 19403.268,E2 19403.268} C_VEL
LIN {X 0,Y 493.701,Z 969.965,A -85,B 0,C 180,E1 19401.793,E2 19401.793} C_VEL
LIN {X 0,Y 488.106,Z 990.401,A -85,B 0,C 180,E1 19400.463,E2 19400.463} C_VEL
LIN {X 0,Y 482.748,Z 1008.629,A -85,B 0,C 180,E1 19399.111,E2 19399.111} C_VEL
LIN {X 0,Y 477.245,Z 1026.315,A -85,B 0,C 180,E1 19397.626,E2 19397.626} C_VEL
LIN {X 0,Y 471.132,Z 1045.123,A -85,B 0,C 180,E1 19395.833,E2 19395.833} C_VEL
LIN {X 0,Y 463.438,Z 1067.803,A -85,B 0,C 180,E1 19393.32,E2 19393.32} C_VEL
LIN {X 0,Y 457.641,Z 1084.314,A -85,B 0,C 180,E1 19391.202,E2 19391.202} C_VEL
LIN {X 0,Y 452.631,Z 1098.477,A -85,B 0,C 180,E1 19389.16,E2 19389.16} C_VEL
LIN {X 0,Y 447.715,Z 1112.369,A -85,B 0,C 180,E1 19386.914,E2 19386.914} C_VEL
LIN {X 0,Y 442.861,Z 1126.36,A -85,B 0,C 180,E1 19384.363,E2 19384.363} C_VEL
LIN {X 0,Y 437.424,Z 1142.523,A -85,B 0,C 180,E1 19380.951,E2 19380.951} C_VEL
LIN {X 0,Y 433.711,Z 1154.283,A -85,B 0,C 180,E1 19378.053,E2 19378.053} C_VEL
LIN {X 0,Y 430.973,Z 1163.69,A -85,B 0,C 180,E1 19375.417,E2 19375.417} C_VEL
LIN {X 0,Y 428.674,Z 1172.395,A -85,B 0,C 180,E1 19372.635,E2 19372.635} C_VEL
LIN {X 0,Y 426.854,Z 1180.421,A -85,B 0,C 180,E1 19369.665,E2 19369.665} C_VEL
LIN {X 0,Y 425.273,Z 1189.004,A -85,B 0,C 180,E1 19365.827,E2 19365.827} C_VEL
LIN {X 0,Y 424.493,Z 1194.59,A -85,B 0,C 180,E1 19362.653,E2 19362.653} C_VEL
LIN {X 0,Y 424.133,Z 1198.597,A -85,B 0,C 180,E1 19359.772,E2 19359.772} C_VEL
LIN {X 0,Y 423.972,Z 1201.447,A -85,B 0,C 180,E1 19357.044,E2 19357.044} C_VEL
LIN {X 0,Y 423.918,Z 1203.369,A -85,B 0,C 180,E1 19354.329,E2 19354.329} C_VEL
LIN {X 0,Y 423.91,Z 1204.373,A -85,B 0,C 180,E1 19351.622,E2 19351.622} C_VEL
LIN {X 0,Y 423.911,Z 1204.463,A -85,B 0,C 180,E1 19348.919,E2 19348.919} C_VEL
LIN {X 0,Y 423.915,Z 1203.639,A -85,B 0,C 180,E1 19346.213,E2 19346.213} C_VEL
LIN {X 0,Y 423.959,Z 1201.898,A -85,B 0,C 180,E1 19343.5,E2 19343.5} C_VEL
LIN {X 0,Y 424.087,Z 1199.23,A -85,B 0,C 180,E1 19340.774,E2 19340.774} C_VEL
LIN {X 0,Y 424.383,Z 1195.618,A -85,B 0,C 180,E1 19338.034,E2 19338.034} C_VEL
LIN {X 0,Y 424.987,Z 1190.78,A -85,B 0,C 180,E1 19335.141,E2 19335.141} C_VEL
LIN {X 0,Y 425.958,Z 1184.846,A -85,B 0,C 180,E1 19332.233,E2 19332.233} C_VEL
LIN {X 0,Y 427.583,Z 1177.077,A -85,B 0,C 180,E1 19329.036,E2 19329.036} C_VEL
LIN {X 0,Y 430.482,Z 1165.642,A -85,B 0,C 180,E1 19325.14,E2 19325.14} C_VEL
LIN {X 0,Y 433.418,Z 1155.568,A -85,B 0,C 180,E1 19322.225,E2 19322.225} C_VEL
LIN {X 0,Y 436.919,Z 1144.717,A -85,B 0,C 180,E1 19319.467,E2 19319.467} C_VEL
LIN {X 0,Y 441.083,Z 1132.544,A -85,B 0,C 180,E1 19316.731,E2 19316.731} C_VEL
LIN {X 0,Y 447.4,Z 1115.233,A -85,B 0,C 180,E1 19313.366,E2 19313.366} C_VEL
LIN {X 0,Y 452.967,Z 1100.255,A -85,B 0,C 180,E1 19310.854,E2 19310.854} C_VEL
LIN {X 0,Y 458.742,Z 1084.886,A -85,B 0,C 180,E1 19308.573,E2 19308.573} C_VEL
LIN {X 0,Y 464.731,Z 1068.921,A -85,B 0,C 180,E1 19306.475,E2 19306.475} C_VEL
LIN {X 0,Y 472.451,Z 1047.981,A -85,B 0,C 180,E1 19304.07,E2 19304.07} C_VEL
LIN {X 0,Y 479.566,Z 1027.639,A -85,B 0,C 180,E1 19302.078,E2 19302.078} C_VEL
LIN {X 0,Y 485.803,Z 1009.115,A -85,B 0,C 180,E1 19300.493,E2 19300.493} C_VEL
LIN {X 0,Y 491.641,Z 990.813,A -85,B 0,C 180,E1 19299.117,E2 19299.117} C_VEL
LIN {X 0,Y 497.474,Z 971.236,A -85,B 0,C 180,E1 19297.826,E2 19297.826} C_VEL
LIN {X 0,Y 504.528,Z 945.184,A -85,B 0,C 180,E1 19296.362,E2 19296.362} C_VEL
LIN {X 0,Y 509.829,Z 922.968,A -85,B 0,C 180,E1 19295.329,E2 19295.329} C_VEL
LIN {X 0,Y 514.204,Z 902.315,A -85,B 0,C 180,E1 19294.516,E2 19294.516} C_VEL
LIN {X 0,Y 518.103,Z 881.296,A -85,B 0,C 180,E1 19293.826,E2 19293.826} C_VEL
LIN {X 0,Y 521.468,Z 859.742,A -85,B 0,C 180,E1 19293.245,E2 19293.245} C_VEL
LIN {X 0,Y 524.866,Z 832.389,A -85,B 0,C 180,E1 19292.674,E2 19292.674} C_VEL
LIN {X 0,Y 527.938,Z 787.358,A -85,B 0,C 180,E1 19291.948,E2 19291.948} C_VEL
LIN {X 0,Y 541.939,Z 564.782,A -85,B 0,C 180,E1 19288.484,E2 19288.484} C_VEL
LIN {X 0,Y 546.198,Z 499.165,A -85,B 0,C 180,E1 19287.443,E2 19287.443} C_VEL
LIN {X 0,Y 538.878,Z 487.296,A -85,B 0,C 180,E1 19285.292,E2 19285.292} C_VEL
LIN {X 0,Y 530.097,Z 473.773,A -85,B 0,C 180,E1 19282.339,E2 19282.339} C_VEL
LIN {X 0,Y 524.006,Z 465.472,A -85,B 0,C 180,E1 19279.972,E2 19279.972} C_VEL
LIN {X 0,Y 520.224,Z 460.5,A -85,B 0,C 180,E1 19278.295,E2 19278.295} C_VEL
LIN {X 0,Y 516.323,Z 455.273,A -85,B 0,C 180,E1 19276.308,E2 19276.308} C_VEL
LIN {X 0,Y 512.988,Z 451.247,A -85,B 0,C 180,E1 19274.332,E2 19274.332} C_VEL
LIN {X 0,Y 512.029,Z 449.804,A -85,B 0,C 180,E1 19273.668,E2 19273.668} C_VEL
LIN {X 0,Y 508.618,Z 445.865,A -85,B 0,C 180,E1 19270.936,E2 19270.936} C_VEL
LIN {X 0,Y 507.667,Z 443.926,A -85,B 0,C 180,E1 19269.867,E2 19269.867} C_VEL
LIN {X 0,Y 504.698,Z 441.599,A -85,B 0,C 180,E1 19264.204,E2 19264.204} C_VEL
LIN {X 0,Y 504.976,Z 441.917,A -85,B 0,C 180,E1 19261.248,E2 19261.248} C_VEL
LIN {X 0,Y 507.903,Z 444.195,A -85,B 0,C 180,E1 19256.671,E2 19256.671} C_VEL
LIN {X 0,Y 510.142,Z 448.095,A -85,B 0,C 180,E1 19254.489,E2 19254.489} C_VEL
LIN {X 0,Y 512.551,Z 450.424,A -85,B 0,C 180,E1 19252.771,E2 19252.771} C_VEL
LIN {X 0,Y 515.639,Z 454.667,A -85,B 0,C 180,E1 19250.851,E2 19250.851} C_VEL
LIN {X 0,Y 517.151,Z 456.408,A -85,B 0,C 180,E1 19250.035,E2 19250.035} C_VEL
LIN {X 0,Y 521.566,Z 462.237,A -85,B 0,C 180,E1 19247.882,E2 19247.882} C_VEL
LIN {X 0,Y 525.951,Z 468.08,A -85,B 0,C 180,E1 19246.028,E2 19246.028} C_VEL
LIN {X 0,Y 530.089,Z 473.644,A -85,B 0,C 180,E1 19244.464,E2 19244.464} C_VEL
LIN {X 0,Y 536.139,Z 481.856,A -85,B 0,C 180,E1 19242.414,E2 19242.414} C_VEL
LIN {X 0,Y 545.255,Z 495.148,A -85,B 0,C 180,E1 19239.693,E2 19239.693} C_VEL
LIN {X 0,Y 546.279,Z 497.101,A -85,B 0,C 180,E1 19239.397,E2 19239.397} C_VEL
LIN {X 0,Y 531.852,Z 720.79,A -85,B 0,C 180,E1 19235.915,E2 19235.915} C_VEL
LIN {X 0,Y 525.568,Z 819.913,A -85,B 0,C 180,E1 19234.358,E2 19234.358} C_VEL
LIN {X 0,Y 522.607,Z 847.553,A -85,B 0,C 180,E1 19233.82,E2 19233.82} C_VEL
LIN {X 0,Y 518.725,Z 873.166,A -85,B 0,C 180,E1 19233.144,E2 19233.144} C_VEL
LIN {X 0,Y 514.861,Z 894.375,A -85,B 0,C 180,E1 19232.451,E2 19232.451} C_VEL
LIN {X 0,Y 510.649,Z 914.596,A -85,B 0,C 180,E1 19231.657,E2 19231.657} C_VEL
LIN {X 0,Y 505.682,Z 935.657,A -85,B 0,C 180,E1 19230.687,E2 19230.687} C_VEL
LIN {X 0,Y 499.224,Z 960.305,A -85,B 0,C 180,E1 19229.34,E2 19229.34} C_VEL
LIN {X 0,Y 492.443,Z 983.074,A -85,B 0,C 180,E1 19227.852,E2 19227.852} C_VEL
LIN {X 0,Y 486.742,Z 1000.941,A -85,B 0,C 180,E1 19226.512,E2 19226.512} C_VEL
LIN {X 0,Y 480.562,Z 1019.23,A -85,B 0,C 180,E1 19224.952,E2 19224.952} C_VEL
LIN {X 0,Y 474.099,Z 1037.538,A -85,B 0,C 180,E1 19223.174,E2 19223.174} C_VEL
LIN {X 0,Y 465.959,Z 1059.691,A -85,B 0,C 180,E1 19220.675,E2 19220.675} C_VEL
LIN {X 0,Y 459.525,Z 1076.579,A -85,B 0,C 180,E1 19218.46,E2 19218.46} C_VEL
LIN {X 0,Y 453.871,Z 1091.356,A -85,B 0,C 180,E1 19216.267,E2 19216.267} C_VEL
LIN {X 0,Y 448.477,Z 1105.526,A -85,B 0,C 180,E1 19213.896,E2 19213.896} C_VEL
LIN {X 0,Y 442.422,Z 1121.872,A -85,B 0,C 180,E1 19210.778,E2 19210.778} C_VEL
LIN {X 0,Y 437.396,Z 1135.946,A -85,B 0,C 180,E1 19207.614,E2 19207.614} C_VEL
LIN {X 0,Y 433.821,Z 1146.696,A -85,B 0,C 180,E1 19204.861,E2 19204.861} C_VEL
LIN {X 0,Y 430.785,Z 1156.668,A -85,B 0,C 180,E1 19201.951,E2 19201.951} C_VEL
LIN {X 0,Y 427.959,Z 1167.374,A -85,B 0,C 180,E1 19198.312,E2 19198.312} C_VEL
LIN {X 0,Y 426.099,Z 1175.741,A -85,B 0,C 180,E1 19194.836,E2 19194.836} C_VEL
LIN {X 0,Y 425.084,Z 1181.541,A -85,B 0,C 180,E1 19191.962,E2 19191.962} C_VEL
LIN {X 0,Y 424.455,Z 1186.268,A -85,B 0,C 180,E1 19189.113,E2 19189.113} C_VEL
LIN {X 0,Y 424.108,Z 1190.122,A -85,B 0,C 180,E1 19186.152,E2 19186.152} C_VEL
LIN {X 0,Y 424.081,Z 1190.583,A -85,B 0,C 180,E1 19185.755,E2 19185.755} C_VEL
LIN {X 0,Y 423.024,Z 1191.7,A -85,B 0,C 180,E1 19184.726,E2 19184.726} C_VEL
LIN {X 0,Y 416.467,Z 1194.002,A -85,B 0,C 180,E1 19181.815,E2 19181.815} C_VEL
LIN {X 0,Y 415.921,Z 1194.363,A -85,B 0,C 180,E1 19181.051,E2 19181.051} C_VEL
LIN {X 0,Y 415.914,Z 1195.241,A -85,B 0,C 180,E1 19178.293,E2 19178.293} C_VEL
LIN {X 0,Y 415.916,Z 1195.224,A -85,B 0,C 180,E1 19175.518,E2 19175.518} C_VEL
LIN {X 0,Y 415.922,Z 1194.309,A -85,B 0,C 180,E1 19172.756,E2 19172.756} C_VEL
LIN {X 0,Y 415.997,Z 1192.393,A -85,B 0,C 180,E1 19169.862,E2 19169.862} C_VEL
LIN {X 0,Y 416.18,Z 1189.501,A -85,B 0,C 180,E1 19166.97,E2 19166.97} C_VEL
LIN {X 0,Y 416.64,Z 1185.221,A -85,B 0,C 180,E1 19163.8,E2 19163.8} C_VEL
LIN {X 0,Y 417.751,Z 1178.367,A -85,B 0,C 180,E1 19159.938,E2 19159.938} C_VEL
LIN {X 0,Y 419.345,Z 1170.912,A -85,B 0,C 180,E1 19156.617,E2 19156.617} C_VEL
LIN {X 0,Y 421.269,Z 1163.284,A -85,B 0,C 180,E1 19153.736,E2 19153.736} C_VEL
LIN {X 0,Y 423.812,Z 1154.463,A -85,B 0,C 180,E1 19150.857,E2 19150.857} C_VEL
LIN {X 0,Y 427.528,Z 1142.914,A -85,B 0,C 180,E1 19147.592,E2 19147.592} C_VEL
LIN {X 0,Y 432.379,Z 1128.845,A -85,B 0,C 180,E1 19144.231,E2 19144.231} C_VEL
LIN {X 0,Y 436.978,Z 1116.069,A -85,B 0,C 180,E1 19141.58,E2 19141.58} C_VEL
LIN {X 0,Y 441.714,Z 1103.273,A -85,B 0,C 180,E1 19139.232,E2 19139.232} C_VEL
LIN {X 0,Y 447.328,Z 1088.278,A -85,B 0,C 180,E1 19136.796,E2 19136.796} C_VEL
LIN {X 0,Y 454.958,Z 1067.714,A -85,B 0,C 180,E1 19133.915,E2 19133.915} C_VEL
LIN {X 0,Y 461.169,Z 1050.481,A -85,B 0,C 180,E1 19131.837,E2 19131.837} C_VEL
LIN {X 0,Y 467.062,Z 1033.633,A -85,B 0,C 180,E1 19130.043,E2 19130.043} C_VEL
LIN {X 0,Y 473.332,Z 1014.929,A -85,B 0,C 180,E1 19128.287,E2 19128.287} C_VEL
LIN {X 0,Y 481.133,Z 990.107,A -85,B 0,C 180,E1 19126.293,E2 19126.293} C_VEL
LIN {X 0,Y 486.971,Z 969.752,A -85,B 0,C 180,E1 19124.899,E2 19124.899} C_VEL
LIN {X 0,Y 492.085,Z 950.51,A -85,B 0,C 180,E1 19123.753,E2 19123.753} C_VEL
LIN {X 0,Y 496.845,Z 930.844,A -85,B 0,C 180,E1 19122.733,E2 19122.733} C_VEL
LIN {X 0,Y 501.655,Z 908.759,A -85,B 0,C 180,E1 19121.753,E2 19121.753} C_VEL
LIN {X 0,Y 506.887,Z 880.318,A -85,B 0,C 180,E1 19120.727,E2 19120.727} C_VEL
LIN {X 0,Y 510.303,Z 857.677,A -85,B 0,C 180,E1 19120.082,E2 19120.082} C_VEL
LIN {X 0,Y 512.928,Z 836.229,A -85,B 0,C 180,E1 19119.595,E2 19119.595} C_VEL
LIN {X 0,Y 514.972,Z 813.165,A -85,B 0,C 180,E1 19119.179,E2 19119.179} C_VEL
LIN {X 0,Y 527.124,Z 597.104,A -85,B 0,C 180,E1 19115.844,E2 19115.844} C_VEL
LIN {X 0,Y 532.846,Z 497.778,A -85,B 0,C 180,E1 19114.297,E2 19114.297} C_VEL
LIN {X 0,Y 523.377,Z 483.815,A -85,B 0,C 180,E1 19112.048,E2 19112.048} C_VEL
LIN {X 0,Y 514.571,Z 471.282,A -85,B 0,C 180,E1 19109.735,E2 19109.735} C_VEL
LIN {X 0,Y 506.008,Z 459.671,A -85,B 0,C 180,E1 19107.223,E2 19107.223} C_VEL
LIN {X 0,Y 499.264,Z 450.823,A -85,B 0,C 180,E1 19104.997,E2 19104.997} C_VEL
LIN {X 0,Y 495.316,Z 445.78,A -85,B 0,C 180,E1 19103.56,E2 19103.56} C_VEL
LIN {X 0,Y 491.22,Z 440.597,A -85,B 0,C 180,E1 19101.933,E2 19101.933} C_VEL
LIN {X 0,Y 487.43,Z 435.589,A -85,B 0,C 180,E1 19100.253,E2 19100.253} C_VEL
LIN {X 0,Y 483.491,Z 431.065,A -85,B 0,C 180,E1 19098.321,E2 19098.321} C_VEL
LIN {X 0,Y 482.436,Z 429.578,A -85,B 0,C 180,E1 19097.738,E2 19097.738} C_VEL
LIN {X 0,Y 479.218,Z 426.327,A -85,B 0,C 180,E1 19095.863,E2 19095.863} C_VEL
LIN {X 0,Y 477.627,Z 423.62,A -85,B 0,C 180,E1 19094.729,E2 19094.729} C_VEL
LIN {X 0,Y 474.474,Z 420.925,A -85,B 0,C 180,E1 19092.289,E2 19092.289} C_VEL
LIN {X 0,Y 472.656,Z 417.375,A -85,B 0,C 180,E1 19090.236,E2 19090.236} C_VEL
LIN {X 0,Y 469.742,Z 415.668,A -85,B 0,C 180,E1 19084.15,E2 19084.15} C_VEL
LIN {X 0,Y 470.405,Z 416.238,A -85,B 0,C 180,E1 19080.244,E2 19080.244} C_VEL
LIN {X 0,Y 472.873,Z 417.671,A -85,B 0,C 180,E1 19076.606,E2 19076.606} C_VEL
LIN {X 0,Y 474.881,Z 421.47,A -85,B 0,C 180,E1 19074.442,E2 19074.442} C_VEL
LIN {X 0,Y 477.975,Z 424.109,A -85,B 0,C 180,E1 19072.124,E2 19072.124} C_VEL
LIN {X 0,Y 480.54,Z 427.931,A -85,B 0,C 180,E1 19070.418,E2 19070.418} C_VEL
LIN {X 0,Y 482.967,Z 430.12,A -85,B 0,C 180,E1 19069.08,E2 19069.08} C_VEL
LIN {X 0,Y 486.325,Z 434.614,A -85,B 0,C 180,E1 19067.352,E2 19067.352} C_VEL
LIN {X 0,Y 487.803,Z 436.266,A -85,B 0,C 180,E1 19066.667,E2 19066.667} C_VEL
LIN {X 0,Y 491.574,Z 440.92,A -85,B 0,C 180,E1 19065.029,E2 19065.029} C_VEL
LIN {X 0,Y 497.146,Z 448.111,A -85,B 0,C 180,E1 19062.863,E2 19062.863} C_VEL
LIN {X 0,Y 501.905,Z 454.317,A -85,B 0,C 180,E1 19061.202,E2 19061.202} C_VEL
LIN {X 0,Y 508.422,Z 462.715,A -85,B 0,C 180,E1 19059.147,E2 19059.147} C_VEL
LIN {X 0,Y 515.741,Z 473.317,A -85,B 0,C 180,E1 19057.035,E2 19057.035} C_VEL
LIN {X 0,Y 526.164,Z 489.545,A -85,B 0,C 180,E1 19054.324,E2 19054.324} C_VEL
LIN {X 0,Y 532.848,Z 500.741,A -85,B 0,C 180,E1 19052.728,E2 19052.728} C_VEL
LIN {X 0,Y 520.576,Z 715.689,A -85,B 0,C 180,E1 19049.409,E2 19049.409} C_VEL
LIN {X 0,Y 514.333,Z 825.712,A -85,B 0,C 180,E1 19047.699,E2 19047.699} C_VEL
LIN {X 0,Y 511.564,Z 853.372,A -85,B 0,C 180,E1 19047.167,E2 19047.167} C_VEL
LIN {X 0,Y 507.8,Z 879.475,A -85,B 0,C 180,E1 19046.485,E2 19046.485} C_VEL
LIN {X 0,Y 504.128,Z 900.735,A -85,B 0,C 180,E1 19045.797,E2 19045.797} C_VEL
LIN {X 0,Y 500.092,Z 921.157,A -85,B 0,C 180,E1 19045.003,E2 19045.003} C_VEL
LIN {X 0,Y 495.305,Z 942.567,A -85,B 0,C 180,E1 19044.023,E2 19044.023} C_VEL
LIN {X 0,Y 488.693,Z 968.951,A -85,B 0,C 180,E1 19042.578,E2 19042.578} C_VEL
LIN {X 0,Y 482.839,Z 989.751,A -85,B 0,C 180,E1 19041.228,E2 19041.228} C_VEL
LIN {X 0,Y 477.303,Z 1008.053,A -85,B 0,C 180,E1 19039.872,E2 19039.872} C_VEL
LIN {X 0,Y 471.349,Z 1026.638,A -85,B 0,C 180,E1 19038.304,E2 19038.304} C_VEL
LIN {X 0,Y 464.892,Z 1045.895,A -85,B 0,C 180,E1 19036.452,E2 19036.452} C_VEL
LIN {X 0,Y 457.113,Z 1067.99,A -85,B 0,C 180,E1 19033.974,E2 19033.974} C_VEL
LIN {X 0,Y 451.137,Z 1084.429,A -85,B 0,C 180,E1 19031.844,E2 19031.844} C_VEL
LIN {X 0,Y 445.748,Z 1099.102,A -85,B 0,C 180,E1 19029.699,E2 19029.699} C_VEL
LIN {X 0,Y 440.429,Z 1113.604,A -85,B 0,C 180,E1 19027.311,E2 19027.311} C_VEL
LIN {X 0,Y 434.425,Z 1130.272,A -85,B 0,C 180,E1 19024.165,E2 19024.165} C_VEL
LIN {X 0,Y 429.61,Z 1144.056,A -85,B 0,C 180,E1 19021.109,E2 19021.109} C_VEL
LIN {X 0,Y 425.978,Z 1155.142,A -85,B 0,C 180,E1 19018.303,E2 19018.303} C_VEL
LIN {X 0,Y 422.994,Z 1165.032,A -85,B 0,C 180,E1 19015.446,E2 19015.446} C_VEL
LIN {X 0,Y 420.116,Z 1175.891,A -85,B 0,C 180,E1 19011.794,E2 19011.794} C_VEL
LIN {X 0,Y 418.2,Z 1184.278,A -85,B 0,C 180,E1 19008.34,E2 19008.34} C_VEL
LIN {X 0,Y 417.15,Z 1190.195,A -85,B 0,C 180,E1 19005.429,E2 19005.429} C_VEL
LIN {X 0,Y 416.488,Z 1194.919,A -85,B 0,C 180,E1 19002.619,E2 19002.619} C_VEL
LIN {X 0,Y 416.138,Z 1198.67,A -85,B 0,C 180,E1 18999.822,E2 18999.822} C_VEL
LIN {X 0,Y 415.972,Z 1201.475,A -85,B 0,C 180,E1 18997.041,E2 18997.041} C_VEL
LIN {X 0,Y 415.918,Z 1203.35,A -85,B 0,C 180,E1 18994.274,E2 18994.274} C_VEL
LIN {X 0,Y 415.912,Z 1204.308,A -85,B 0,C 180,E1 18991.515,E2 18991.515} C_VEL
LIN {X 0,Y 415.912,Z 1204.375,A -85,B 0,C 180,E1 18988.898,E2 18988.898} C_VEL
LIN {X 0,Y 415.915,Z 1203.535,A -85,B 0,C 180,E1 18986.109,E2 18986.109} C_VEL
LIN {X 0,Y 415.961,Z 1201.809,A -85,B 0,C 180,E1 18983.375,E2 18983.375} C_VEL
LIN {X 0,Y 416.1,Z 1199.14,A -85,B 0,C 180,E1 18980.596,E2 18980.596} C_VEL
LIN {X 0,Y 416.443,Z 1195.317,A -85,B 0,C 180,E1 18977.662,E2 18977.662} C_VEL
LIN {X 0,Y 417.066,Z 1190.691,A -85,B 0,C 180,E1 18974.852,E2 18974.852} C_VEL
LIN {X 0,Y 418.102,Z 1184.771,A -85,B 0,C 180,E1 18971.887,E2 18971.887} C_VEL
LIN {X 0,Y 419.753,Z 1177.378,A -85,B 0,C 180,E1 18968.773,E2 18968.773} C_VEL
LIN {X 0,Y 422.662,Z 1166.542,A -85,B 0,C 180,E1 18964.948,E2 18964.948} C_VEL
LIN {X 0,Y 426.028,Z 1155.574,A -85,B 0,C 180,E1 18961.701,E2 18961.701} C_VEL
LIN {X 0,Y 429.702,Z 1144.752,A -85,B 0,C 180,E1 18958.898,E2 18958.898} C_VEL
LIN {X 0,Y 434.085,Z 1132.606,A -85,B 0,C 180,E1 18956.123,E2 18956.123} C_VEL
LIN {X 0,Y 440.477,Z 1115.959,A -85,B 0,C 180,E1 18952.824,E2 18952.824} C_VEL
LIN {X 0,Y 446.508,Z 1100.404,A -85,B 0,C 180,E1 18950.176,E2 18950.176} C_VEL
LIN {X 0,Y 452.314,Z 1085.6,A -85,B 0,C 180,E1 18947.949,E2 18947.949} C_VEL
LIN {X 0,Y 458.456,Z 1069.875,A -85,B 0,C 180,E1 18945.853,E2 18945.853} C_VEL
LIN {X 0,Y 465.412,Z 1051.767,A -85,B 0,C 180,E1 18943.726,E2 18943.726} C_VEL
LIN {X 0,Y 473.879,Z 1028.65,A -85,B 0,C 180,E1 18941.402,E2 18941.402} C_VEL
LIN {X 0,Y 480.539,Z 1009.513,A -85,B 0,C 180,E1 18939.752,E2 18939.752} C_VEL
LIN {X 0,Y 486.809,Z 990.477,A -85,B 0,C 180,E1 18938.317,E2 18938.317} C_VEL
LIN {X 0,Y 492.833,Z 970.885,A -85,B 0,C 180,E1 18937.029,E2 18937.029} C_VEL
LIN {X 0,Y 499.984,Z 945.19,A -85,B 0,C 180,E1 18935.588,E2 18935.588} C_VEL
LIN {X 0,Y 505.54,Z 922.521,A -85,B 0,C 180,E1 18934.538,E2 18934.538} C_VEL
LIN {X 0,Y 510.054,Z 901.756,A -85,B 0,C 180,E1 18933.726,E2 18933.726} C_VEL
LIN {X 0,Y 514.018,Z 880.845,A -85,B 0,C 180,E1 18933.044,E2 18933.044} C_VEL
LIN {X 0,Y 517.528,Z 858.832,A -85,B 0,C 180,E1 18932.457,E2 18932.457} C_VEL
LIN {X 0,Y 521.033,Z 830.414,A -85,B 0,C 180,E1 18931.876,E2 18931.876} C_VEL
LIN {X 0,Y 524.327,Z 782.801,A -85,B 0,C 180,E1 18931.111,E2 18931.111} C_VEL
LIN {X 0,Y 538.69,Z 561.79,A -85,B 0,C 180,E1 18927.667,E2 18927.667} C_VEL
LIN {X 0,Y 542.571,Z 504.036,A -85,B 0,C 180,E1 18926.755,E2 18926.755} C_VEL
LIN {X 0,Y 536.264,Z 493.729,A -85,B 0,C 180,E1 18924.834,E2 18924.834} C_VEL
LIN {X 0,Y 528.121,Z 480.961,A -85,B 0,C 180,E1 18922.017,E2 18922.017} C_VEL
LIN {X 0,Y 522.403,Z 473.033,A -85,B 0,C 180,E1 18919.744,E2 18919.744} C_VEL
LIN {X 0,Y 518.608,Z 468.006,A -85,B 0,C 180,E1 18918.026,E2 18918.026} C_VEL
LIN {X 0,Y 514.752,Z 462.81,A -85,B 0,C 180,E1 18916.012,E2 18916.012} C_VEL
LIN {X 0,Y 511.526,Z 458.667,A -85,B 0,C 180,E1 18914.027,E2 18914.027} C_VEL
LIN {X 0,Y 510.736,Z 457.572,A -85,B 0,C 180,E1 18913.472,E2 18913.472} C_VEL
LIN {X 0,Y 507.369,Z 453.465,A -85,B 0,C 180,E1 18910.676,E2 18910.676} C_VEL
LIN {X 0,Y 506.592,Z 451.831,A -85,B 0,C 180,E1 18909.773,E2 18909.773} C_VEL
LIN {X 0,Y 503.71,Z 449.523,A -85,B 0,C 180,E1 18904.098,E2 18904.098} C_VEL
LIN {X 0,Y 504.065,Z 449.969,A -85,B 0,C 180,E1 18901.023,E2 18901.023} C_VEL
LIN {X 0,Y 506.809,Z 452.12,A -85,B 0,C 180,E1 18896.777,E2 18896.777} C_VEL
LIN {X 0,Y 509.156,Z 456.126,A -85,B 0,C 180,E1 18894.478,E2 18894.478} C_VEL
LIN {X 0,Y 511.312,Z 458.249,A -85,B 0,C 180,E1 18892.923,E2 18892.923} C_VEL
LIN {X 0,Y 514.458,Z 462.549,A -85,B 0,C 180,E1 18890.942,E2 18890.942} C_VEL
LIN {X 0,Y 515.747,Z 464.098,A -85,B 0,C 180,E1 18890.233,E2 18890.233} C_VEL
LIN {X 0,Y 520.092,Z 469.94,A -85,B 0,C 180,E1 18888.073,E2 18888.073} C_VEL
LIN {X 0,Y 524.417,Z 475.795,A -85,B 0,C 180,E1 18886.212,E2 18886.212} C_VEL
LIN {X 0,Y 528.791,Z 481.767,A -85,B 0,C 180,E1 18884.537,E2 18884.537} C_VEL
LIN {X 0,Y 534.796,Z 490.151,A -85,B 0,C 180,E1 18882.481,E2 18882.481} C_VEL
LIN {X 0,Y 542.644,Z 501.719,A -85,B 0,C 180,E1 18880.097,E2 18880.097} C_VEL
LIN {X 0,Y 527.927,Z 723.372,A -85,B 0,C 180,E1 18876.643,E2 18876.643} C_VEL
LIN {X 0,Y 521.592,Z 820.104,A -85,B 0,C 180,E1 18875.119,E2 18875.119} C_VEL
LIN {X 0,Y 518.54,Z 847.832,A -85,B 0,C 180,E1 18874.58,E2 18874.58} C_VEL
LIN {X 0,Y 514.585,Z 873.293,A -85,B 0,C 180,E1 18873.91,E2 18873.91} C_VEL
LIN {X 0,Y 510.671,Z 894.261,A -85,B 0,C 180,E1 18873.229,E2 18873.229} C_VEL
LIN {X 0,Y 506.225,Z 915.02,A -85,B 0,C 180,E1 18872.416,E2 18872.416} C_VEL
LIN {X 0,Y 501.276,Z 935.429,A -85,B 0,C 180,E1 18871.477,E2 18871.477} C_VEL
LIN {X 0,Y 494.634,Z 960.135,A -85,B 0,C 180,E1 18870.133,E2 18870.133} C_VEL
LIN {X 0,Y 487.619,Z 982.994,A -85,B 0,C 180,E1 18868.641,E2 18868.641} C_VEL
LIN {X 0,Y 481.502,Z 1001.549,A -85,B 0,C 180,E1 18867.245,E2 18867.245} C_VEL
LIN {X 0,Y 475.394,Z 1019.06,A -85,B 0,C 180,E1 18865.747,E2 18865.747} C_VEL
LIN {X 0,Y 468.9,Z 1036.828,A -85,B 0,C 180,E1 18864.02,E2 18864.02} C_VEL
LIN {X 0,Y 461.092,Z 1057.47,A -85,B 0,C 180,E1 18861.719,E2 18861.719} C_VEL
LIN {X 0,Y 453.698,Z 1076.065,A -85,B 0,C 180,E1 18859.281,E2 18859.281} C_VEL
LIN {X 0,Y 447.793,Z 1090.864,A -85,B 0,C 180,E1 18857.074,E2 18857.074} C_VEL
LIN {X 0,Y 442.153,Z 1105.024,A -85,B 0,C 180,E1 18854.69,E2 18854.69} C_VEL
LIN {X 0,Y 436.33,Z 1120.012,A -85,B 0,C 180,E1 18851.823,E2 18851.823} C_VEL
LIN {X 0,Y 430.665,Z 1134.976,A -85,B 0,C 180,E1 18848.477,E2 18848.477} C_VEL
LIN {X 0,Y 426.65,Z 1146.355,A -85,B 0,C 180,E1 18845.534,E2 18845.534} C_VEL
LIN {X 0,Y 423.545,Z 1155.887,A -85,B 0,C 180,E1 18842.724,E2 18842.724} C_VEL
LIN {X 0,Y 420.864,Z 1165.136,A -85,B 0,C 180,E1 18839.594,E2 18839.594} C_VEL
LIN {X 0,Y 418.457,Z 1174.919,A -85,B 0,C 180,E1 18835.625,E2 18835.625} C_VEL
LIN {X 0,Y 417.226,Z 1181.376,A -85,B 0,C 180,E1 18832.398,E2 18832.398} C_VEL
LIN {X 0,Y 416.526,Z 1186.143,A -85,B 0,C 180,E1 18829.491,E2 18829.491} C_VEL
LIN {X 0,Y 416.153,Z 1189.883,A -85,B 0,C 180,E1 18826.613,E2 18826.613} C_VEL
LIN {X 0,Y 415.977,Z 1192.629,A -85,B 0,C 180,E1 18823.766,E2 18823.766} C_VEL
LIN {X 0,Y 415.921,Z 1194.363,A -85,B 0,C 180,E1 18821.051,E2 18821.051} C_VEL
LIN {X 0,Y 414.914,Z 1194.904,A -85,B 0,C 180,E1 18819.992,E2 18819.992} C_VEL
LIN {X 0,Y 408.345,Z 1195.533,A -85,B 0,C 180,E1 18816.926,E2 18816.926} C_VEL
LIN {X 0,Y 407.916,Z 1195.427,A -85,B 0,C 180,E1 18816.222,E2 18816.222} C_VEL
LIN {X 0,Y 407.919,Z 1194.66,A -85,B 0,C 180,E1 18813.232,E2 18813.232} C_VEL
LIN {X 0,Y 407.981,Z 1192.92,A -85,B 0,C 180,E1 18810.281,E2 18810.281} C_VEL
LIN {X 0,Y 408.152,Z 1190.205,A -85,B 0,C 180,E1 18807.332,E2 18807.332} C_VEL
LIN {X 0,Y 408.534,Z 1186.505,A -85,B 0,C 180,E1 18804.382,E2 18804.382} C_VEL
LIN {X 0,Y 409.201,Z 1182.048,A -85,B 0,C 180,E1 18801.57,E2 18801.57} C_VEL
LIN {X 0,Y 410.312,Z 1176.36,A -85,B 0,C 180,E1 18798.616,E2 18798.616} C_VEL
LIN {X 0,Y 411.921,Z 1169.605,A -85,B 0,C 180,E1 18795.665,E2 18795.665} C_VEL
LIN {X 0,Y 414.463,Z 1160.556,A -85,B 0,C 180,E1 18792.304,E2 18792.304} C_VEL
LIN {X 0,Y 418.323,Z 1148.38,A -85,B 0,C 180,E1 18788.55,E2 18788.55} C_VEL
LIN {X 0,Y 422.14,Z 1137.437,A -85,B 0,C 180,E1 18785.662,E2 18785.662} C_VEL
LIN {X 0,Y 426.435,Z 1125.713,A -85,B 0,C 180,E1 18782.944,E2 18782.944} C_VEL
LIN {X 0,Y 432.002,Z 1111.232,A -85,B 0,C 180,E1 18780.005,E2 18780.005} C_VEL
LIN {X 0,Y 438.706,Z 1093.863,A -85,B 0,C 180,E1 18776.996,E2 18776.996} C_VEL
LIN {X 0,Y 444.599,Z 1078.584,A -85,B 0,C 180,E1 18774.692,E2 18774.692} C_VEL
LIN {X 0,Y 450.324,Z 1063.578,A -85,B 0,C 180,E1 18772.689,E2 18772.689} C_VEL
LIN {X 0,Y 456.264,Z 1047.6,A -85,B 0,C 180,E1 18770.795,E2 18770.795} C_VEL
LIN {X 0,Y 463.536,Z 1027.437,A -85,B 0,C 180,E1 18768.697,E2 18768.697} C_VEL
LIN {X 0,Y 471.03,Z 1005.014,A -85,B 0,C 180,E1 18766.715,E2 18766.715} C_VEL
LIN {X 0,Y 476.775,Z 986.756,A -85,B 0,C 180,E1 18765.313,E2 18765.313} C_VEL
LIN {X 0,Y 482.161,Z 968.348,A -85,B 0,C 180,E1 18764.066,E2 18764.066} C_VEL
LIN {X 0,Y 487.694,Z 947.885,A -85,B 0,C 180,E1 18762.861,E2 18762.861} C_VEL
LIN {X 0,Y 493.735,Z 923.264,A -85,B 0,C 180,E1 18761.625,E2 18761.625} C_VEL
LIN {X 0,Y 498.998,Z 897.817,A -85,B 0,C 180,E1 18760.588,E2 18760.588} C_VEL
LIN {X 0,Y 502.837,Z 876.298,A -85,B 0,C 180,E1 18759.862,E2 18759.862} C_VEL
LIN {X 0,Y 506.047,Z 854.973,A -85,B 0,C 180,E1 18759.272,E2 18759.272} C_VEL
LIN {X 0,Y 508.872,Z 831.695,A -85,B 0,C 180,E1 18758.764,E2 18758.764} C_VEL
LIN {X 0,Y 511.527,Z 795.808,A -85,B 0,C 180,E1 18758.162,E2 18758.162} C_VEL
LIN {X 0,Y 524.49,Z 571.707,A -85,B 0,C 180,E1 18754.701,E2 18754.701} C_VEL
LIN {X 0,Y 528.564,Z 502.182,A -85,B 0,C 180,E1 18753.602,E2 18753.602} C_VEL
LIN {X 0,Y 518.024,Z 486.64,A -85,B 0,C 180,E1 18750.99,E2 18750.99} C_VEL
LIN {X 0,Y 508.737,Z 473.463,A -85,B 0,C 180,E1 18748.401,E2 18748.401} C_VEL
LIN {X 0,Y 501.102,Z 463.175,A -85,B 0,C 180,E1 18746.007,E2 18746.007} C_VEL
LIN {X 0,Y 496.747,Z 457.46,A -85,B 0,C 180,E1 18744.498,E2 18744.498} C_VEL
LIN {X 0,Y 493.33,Z 453.015,A -85,B 0,C 180,E1 18743.217,E2 18743.217} C_VEL
LIN {X 0,Y 489.447,Z 448.027,A -85,B 0,C 180,E1 18741.638,E2 18741.638} C_VEL
LIN {X 0,Y 485.166,Z 442.554,A -85,B 0,C 180,E1 18739.692,E2 18739.692} C_VEL
LIN {X 0,Y 481.476,Z 437.759,A -85,B 0,C 180,E1 18737.775,E2 18737.775} C_VEL
LIN {X 0,Y 477.715,Z 433.762,A -85,B 0,C 180,E1 18735.54,E2 18735.54} C_VEL
LIN {X 0,Y 476.418,Z 431.463,A -85,B 0,C 180,E1 18734.587,E2 18734.587} C_VEL
LIN {X 0,Y 473.248,Z 428.643,A -85,B 0,C 180,E1 18732.074,E2 18732.074} C_VEL
LIN {X 0,Y 471.582,Z 425.289,A -85,B 0,C 180,E1 18730.136,E2 18730.136} C_VEL
LIN {X 0,Y 468.766,Z 423.608,A -85,B 0,C 180,E1 18724.159,E2 18724.159} C_VEL
LIN {X 0,Y 469.426,Z 424.183,A -85,B 0,C 180,E1 18720.244,E2 18720.244} C_VEL
LIN {X 0,Y 471.78,Z 425.599,A -85,B 0,C 180,E1 18716.72,E2 18716.72} C_VEL
LIN {X 0,Y 473.76,Z 429.343,A -85,B 0,C 180,E1 18714.55,E2 18714.55} C_VEL
LIN {X 0,Y 476.65,Z 431.796,A -85,B 0,C 180,E1 18712.345,E2 18712.345} C_VEL
LIN {X 0,Y 479.36,Z 435.817,A -85,B 0,C 180,E1 18710.515,E2 18710.515} C_VEL
LIN {X 0,Y 481.647,Z 438.006,A -85,B 0,C 180,E1 18709.232,E2 18709.232} C_VEL
LIN {X 0,Y 485.101,Z 442.523,A -85,B 0,C 180,E1 18707.44,E2 18707.44} C_VEL
LIN {X 0,Y 486.667,Z 444.554,A -85,B 0,C 180,E1 18706.696,E2 18706.696} C_VEL
LIN {X 0,Y 490.974,Z 449.92,A -85,B 0,C 180,E1 18704.829,E2 18704.829} C_VEL
LIN {X 0,Y 495.542,Z 455.875,A -85,B 0,C 180,E1 18703.048,E2 18703.048} C_VEL
LIN {X 0,Y 500.095,Z 461.874,A -85,B 0,C 180,E1 18701.433,E2 18701.433} C_VEL
LIN {X 0,Y 506.449,Z 470.219,A -85,B 0,C 180,E1 18699.395,E2 18699.395} C_VEL
LIN {X 0,Y 513.315,Z 480.323,A -85,B 0,C 180,E1 18697.374,E2 18697.374} C_VEL
LIN {X 0,Y 523.399,Z 496.254,A -85,B 0,C 180,E1 18694.694,E2 18694.694} C_VEL
LIN {X 0,Y 528.606,Z 505.102,A -85,B 0,C 180,E1 18693.414,E2 18693.414} C_VEL
LIN {X 0,Y 515.937,Z 720.541,A -85,B 0,C 180,E1 18690.079,E2 18690.079} C_VEL
LIN {X 0,Y 509.777,Z 825.783,A -85,B 0,C 180,E1 18688.437,E2 18688.437} C_VEL
LIN {X 0,Y 506.943,Z 853.386,A -85,B 0,C 180,E1 18687.906,E2 18687.906} C_VEL
LIN {X 0,Y 503.091,Z 879.446,A -85,B 0,C 180,E1 18687.226,E2 18687.226} C_VEL
LIN {X 0,Y 499.403,Z 900.337,A -85,B 0,C 180,E1 18686.551,E2 18686.551} C_VEL
LIN {X 0,Y 495.271,Z 920.734,A -85,B 0,C 180,E1 18685.761,E2 18685.761} C_VEL
LIN {X 0,Y 490.546,Z 941.42,A -85,B 0,C 180,E1 18684.819,E2 18684.819} C_VEL
LIN {X 0,Y 484.309,Z 966.085,A -85,B 0,C 180,E1 18683.492,E2 18683.492} C_VEL
LIN {X 0,Y 477.692,Z 988.962,A -85,B 0,C 180,E1 18682.019,E2 18682.019} C_VEL
LIN {X 0,Y 471.708,Z 1008.213,A -85,B 0,C 180,E1 18680.589,E2 18680.589} C_VEL
LIN {X 0,Y 465.811,Z 1026.106,A -85,B 0,C 180,E1 18679.074,E2 18679.074} C_VEL
LIN {X 0,Y 459.414,Z 1044.593,A -85,B 0,C 180,E1 18677.295,E2 18677.295} C_VEL
LIN {X 0,Y 451.294,Z 1066.996,A -85,B 0,C 180,E1 18674.792,E2 18674.792} C_VEL
LIN {X 0,Y 444.864,Z 1084.051,A -85,B 0,C 180,E1 18672.572,E2 18672.572} C_VEL
LIN {X 0,Y 439.339,Z 1098.562,A -85,B 0,C 180,E1 18670.437,E2 18670.437} C_VEL
LIN {X 0,Y 434.011,Z 1112.507,A -85,B 0,C 180,E1 18668.127,E2 18668.127} C_VEL
LIN {X 0,Y 428.245,Z 1127.962,A -85,B 0,C 180,E1 18665.218,E2 18665.218} C_VEL
LIN {X 0,Y 422.607,Z 1143.245,A -85,B 0,C 180,E1 18661.843,E2 18661.843} C_VEL
LIN {X 0,Y 418.777,Z 1154.417,A -85,B 0,C 180,E1 18658.991,E2 18658.991} C_VEL
LIN {X 0,Y 415.613,Z 1164.28,A -85,B 0,C 180,E1 18656.12,E2 18656.12} C_VEL
LIN {X 0,Y 412.895,Z 1173.742,A -85,B 0,C 180,E1 18652.947,E2 18652.947} C_VEL
LIN {X 0,Y 410.536,Z 1183.419,A -85,B 0,C 180,E1 18649.048,E2 18649.048} C_VEL
LIN {X 0,Y 409.245,Z 1190.087,A -85,B 0,C 180,E1 18645.735,E2 18645.735} C_VEL
LIN {X 0,Y 408.532,Z 1194.822,A -85,B 0,C 180,E1 18642.869,E2 18642.869} C_VEL
LIN {X 0,Y 408.155,Z 1198.602,A -85,B 0,C 180,E1 18639.997,E2 18639.997} C_VEL
LIN {X 0,Y 407.981,Z 1201.387,A -85,B 0,C 180,E1 18637.18,E2 18637.18} C_VEL
LIN {X 0,Y 407.918,Z 1203.263,A -85,B 0,C 180,E1 18634.358,E2 18634.358} C_VEL
LIN {X 0,Y 407.91,Z 1204.198,A -85,B 0,C 180,E1 18631.686,E2 18631.686} C_VEL
LIN {X 0,Y 407.913,Z 1204.288,A -85,B 0,C 180,E1 18628.876,E2 18628.876} C_VEL
LIN {X 0,Y 407.916,Z 1203.462,A -85,B 0,C 180,E1 18626.065,E2 18626.065} C_VEL
LIN {X 0,Y 407.964,Z 1201.72,A -85,B 0,C 180,E1 18623.244,E2 18623.244} C_VEL
LIN {X 0,Y 408.116,Z 1199.052,A -85,B 0,C 180,E1 18620.41,E2 18620.41} C_VEL
LIN {X 0,Y 408.483,Z 1195.236,A -85,B 0,C 180,E1 18617.417,E2 18617.417} C_VEL
LIN {X 0,Y 409.157,Z 1190.621,A -85,B 0,C 180,E1 18614.552,E2 18614.552} C_VEL
LIN {X 0,Y 410.262,Z 1184.715,A -85,B 0,C 180,E1 18611.529,E2 18611.529} C_VEL
LIN {X 0,Y 412.023,Z 1177.332,A -85,B 0,C 180,E1 18608.351,E2 18608.351} C_VEL
LIN {X 0,Y 415.113,Z 1166.539,A -85,B 0,C 180,E1 18604.46,E2 18604.46} C_VEL
LIN {X 0,Y 418.677,Z 1155.597,A -85,B 0,C 180,E1 18601.158,E2 18601.158} C_VEL
LIN {X 0,Y 422.527,Z 1144.799,A -85,B 0,C 180,E1 18598.309,E2 18598.309} C_VEL
LIN {X 0,Y 427.18,Z 1132.611,A -85,B 0,C 180,E1 18595.479,E2 18595.479} C_VEL
LIN {X 0,Y 433.764,Z 1116.243,A -85,B 0,C 180,E1 18592.183,E2 18592.183} C_VEL
LIN {X 0,Y 440.115,Z 1100.564,A -85,B 0,C 180,E1 18589.478,E2 18589.478} C_VEL
LIN {X 0,Y 446.339,Z 1085.342,A -85,B 0,C 180,E1 18587.166,E2 18587.166} C_VEL
LIN {X 0,Y 452.786,Z 1069.469,A -85,B 0,C 180,E1 18585.038,E2 18585.038} C_VEL
LIN {X 0,Y 460.907,Z 1049.17,A -85,B 0,C 180,E1 18582.659,E2 18582.659} C_VEL
LIN {X 0,Y 468.982,Z 1027.665,A -85,B 0,C 180,E1 18580.528,E2 18580.528} C_VEL
LIN {X 0,Y 475.742,Z 1008.841,A -85,B 0,C 180,E1 18578.908,E2 18578.908} C_VEL
LIN {X 0,Y 482.077,Z 990.154,A -85,B 0,C 180,E1 18577.503,E2 18577.503} C_VEL
LIN {X 0,Y 488.844,Z 968.771,A -85,B 0,C 180,E1 18576.108,E2 18576.108} C_VEL
LIN {X 0,Y 496.126,Z 942.93,A -85,B 0,C 180,E1 18574.689,E2 18574.689} C_VEL
LIN {X 0,Y 501.352,Z 922.09,A -85,B 0,C 180,E1 18573.734,E2 18573.734} C_VEL
LIN {X 0,Y 505.854,Z 901.923,A -85,B 0,C 180,E1 18572.949,E2 18572.949} C_VEL
LIN {X 0,Y 509.93,Z 880.976,A -85,B 0,C 180,E1 18572.268,E2 18572.268} C_VEL
LIN {X 0,Y 513.513,Z 859.11,A -85,B 0,C 180,E1 18571.686,E2 18571.686} C_VEL
LIN {X 0,Y 517.084,Z 831.188,A -85,B 0,C 180,E1 18571.113,E2 18571.113} C_VEL
LIN {X 0,Y 520.395,Z 785.012,A -85,B 0,C 180,E1 18570.369,E2 18570.369} C_VEL
LIN {X 0,Y 535.258,Z 563.019,A -85,B 0,C 180,E1 18566.906,E2 18566.906} C_VEL
LIN {X 0,Y 539.013,Z 508.893,A -85,B 0,C 180,E1 18566.052,E2 18566.052} C_VEL
LIN {X 0,Y 532.462,Z 498.094,A -85,B 0,C 180,E1 18563.959,E2 18563.959} C_VEL
LIN {X 0,Y 525.203,Z 486.775,A -85,B 0,C 180,E1 18561.323,E2 18561.323} C_VEL
LIN {X 0,Y 520.559,Z 480.297,A -85,B 0,C 180,E1 18559.408,E2 18559.408} C_VEL
LIN {X 0,Y 517.19,Z 475.706,A -85,B 0,C 180,E1 18557.844,E2 18557.844} C_VEL
LIN {X 0,Y 513.393,Z 470.526,A -85,B 0,C 180,E1 18555.823,E2 18555.823} C_VEL
LIN {X 0,Y 510.155,Z 466.229,A -85,B 0,C 180,E1 18553.777,E2 18553.777} C_VEL
LIN {X 0,Y 508.979,Z 464.945,A -85,B 0,C 180,E1 18552.941,E2 18552.941} C_VEL
LIN {X 0,Y 505.975,Z 460.703,A -85,B 0,C 180,E1 18550.233,E2 18550.233} C_VEL
LIN {X 0,Y 505.414,Z 459.689,A -85,B 0,C 180,E1 18549.566,E2 18549.566} C_VEL
LIN {X 0,Y 502.734,Z 457.466,A -85,B 0,C 180,E1 18544.106,E2 18544.106} C_VEL
LIN {X 0,Y 503.085,Z 457.917,A -85,B 0,C 180,E1 18541.025,E2 18541.025} C_VEL
LIN {X 0,Y 505.717,Z 460.04,A -85,B 0,C 180,E1 18536.883,E2 18536.883} C_VEL
LIN {X 0,Y 508.171,Z 464.154,A -85,B 0,C 180,E1 18534.467,E2 18534.467} C_VEL
LIN {X 0,Y 510.078,Z 466.07,A -85,B 0,C 180,E1 18533.076,E2 18533.076} C_VEL
LIN {X 0,Y 513.278,Z 470.43,A -85,B 0,C 180,E1 18531.034,E2 18531.034} C_VEL
